RoboDK station: Demo-opstelling - Full - test 2 - for approach point generation - production.rdk

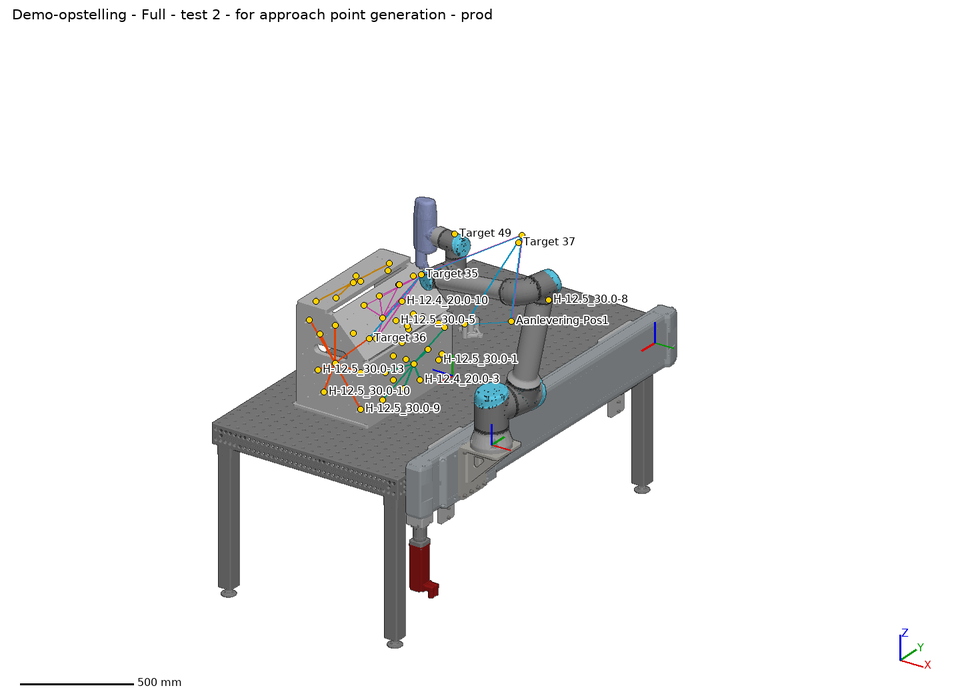
[picture v0: the station drawn from its stored meshes, robots at their saved joint values, targets as dots, program paths as lines]
Station Demo-opstelling - Full - test 2 - Copy (saved by RoboDK 5.9.0). Poses are relative to the parent item; angles as X-Y-Z fixed-axis rotations.
Station parameters (name, value as stored): CollisionFreePlanner, UR10e, CollisionFreePlanner-Rob UR10e, CollisionFreePlanner-Rob My Mechanism, CollisionFreePlanner-Rob Lineaire rail
  - object Lineaire Rail at (0, 0, 0) mm, size 171.1 x 1963 x 635.1 mm
  - object Cobot Carraige at (0, 0, 0) mm, size 240 x 425 x 269.5 mm
  - object Lastafel at (0, 0, 0) mm, size 1021.8 x 2000 x 842 mm
  - frame Lineaire rail  Base at (218.83, 1501.27, 137) mm, rotated rx 0 ry 0 rz -90 deg
    - robot Lineaire rail: 1 axes
        modified DH rows (alpha deg, a mm, theta deg, d mm): 0, 0, 0, 0 linear
        base shift (0, 0, 0) mm, rotated rx 0 ry 90 rz 0 deg
        joint limits [-1248] to [-1248]; home [0]; saved at [-1248]
      - frame UR10e Base at (0, -2, 0.1) mm, rotated rx 0 ry 0 rz 90 deg
        - robot UR10e: 6 axes, payload 10 kg, reach 1300 mm, repeatability 0.05 mm, weight 28.9 kg
            modified DH rows (alpha deg, a mm, theta deg, d mm): 0, 0, 0, 180.7; 90, 0, 180, 0; 0, 612.6, 0, 0; 0, 571.335, 0, 174.15; -90, 0, 0, 119.85; 90, 0, 180, 116.55
            joint limits [100, -200, -360, -480, -360, -360] to [250, 180, 360, 360, 360, 700]; home [30.872, -95.296, 116.362, -22.187, 121.11, 179.827]; saved at [168.209, -76.445, -115.546, 11.991, 92.546, 90.001]
          - tool TCP Schroeftool, TCP at (225, 0, 93) mm, rotated rx 90 ry -90 rz 90 deg, size 86.2 x 125.3 x 346 mm, geometry from Onrobot + custom dop.STEP
          - tool TCP Sensor, TCP at (-192.58, 8.55, 68.16) mm, rotated rx 0 ry -90 rz 0 deg
  - Python program csv_importer_v12 (listed below)
  - program Oppakken (1 instructions, listed below)
  - program indraaien/uitdraaien (1 instructions, listed below)
  - Python program importRobotPoints (listed below)
  - Python program __init__ (listed below)
  - program Prog8 (11 instructions, listed below)
  - frame CSV Frame at (-421.32, 863.78, 53.03) mm, rotated rx 90 ry 0 rz -89.82 deg
    - object Test object at (0, 0, 0) mm, size 650 x 517 x 400 mm, geometry from Test object.STEP
    - target Target 35 (Cartesian target) at (321.7, 636.46, -59.39) mm, rotated rx -90 ry -80.58 rz -180 deg; joints [168.209, -76.49, -91.294, -192.215, -92.546, 270.001] of UR10e
    - target Target 37 (Cartesian target) at (-229.45, 611.91, -197.99) mm, rotated rx 0 ry -0.72 rz 180 deg; joints [123.607, -98.633, -95.414, -165.955, -57.291, 0.002] of UR10e
    - target Target 36 (Cartesian target) at (850.47, 562.22, -149.07) mm, rotated rx 70.72 ry 0 rz -90 deg; joints [244.224, -80.879, -108.983, -80.137, 89.999, 44.77] of UR10e
    - target H-12.5_30.0-0 (Cartesian target) at (10, 165.95, 226.14) mm, rotated rx -90 ry 0 rz -90 deg; joints [161.752, -90.555, -88.742, -182.846, -147.095, -106.726] of UR10e
    - target H-12.5_30.0-1 (Cartesian target) at (10, 61.56, 64.68) mm, rotated rx -90 ry 1.14 rz -90.86 deg; joints [140.207, -149.215, -63.175, -57.939, 88.607, 140.221] of UR10e
    - target H-12.5_30.0-2 (Cartesian target) at (10, 91.63, 261.38) mm, rotated rx -90 ry 0 rz -90 deg; joints [139.629, -149.975, -62.079, -417.947, 89.999, 139.63] of UR10e
    - target H-12.5_30.0-3 (Cartesian target) at (10, 435.06, 200.51) mm, rotated rx -90 ry 0 rz -90 deg; joints [145.332, -190.81, 25.853, -105.043, 89.999, 145.334] of UR10e
    - target H-12.5_30.0-4 (Cartesian target) at (10, 369.06, 279.32) mm, rotated rx -90 ry 0 rz -90 deg; joints [143.714, -169.382, 16.894, 242.486, 89.999, 143.716] of UR10e
    - target H-12.5_30.0-5 (Cartesian target) at (10, 190.3, 292.78) mm, rotated rx -90 ry 0 rz -90 deg; joints [166.618, -153.245, -71.353, -35.667, -87.696, -166.813] of UR10e
    - target H-12.5_30.0-6 (Cartesian target) at (10, 241.56, 64.68) mm, rotated rx -90 ry 0 rz -90 deg; joints [166.782, 132.561, 62.356, 264.825, -87.724, -166.975] of UR10e
    - target H-12.5_30.0-7 (Cartesian target) at (10, 422.89, 336.81) mm, rotated rx -90 ry 0 rz -90 deg; joints [139.629, -141.427, -58.919, -69.655, 89.999, 139.63] of UR10e
    - target H-12.5_30.0-8 (Cartesian target) at (-862.39, -0.19, 81.88) mm, rotated rx 122.16 ry 90 rz -147.65 deg; joints [205.922, -142.466, -64.883, -242.648, -90, -154.261] of UR10e
    - target H-12.5_30.0-9 (Cartesian target) at (610, 61.56, 64.68) mm, rotated rx 90 ry 0 rz -90 deg; joints [202.083, -127.057, -94.792, -48.15, 90, 22.085] of UR10e
    - target H-12.5_30.0-10 (Cartesian target) at (610, 91.63, 261.38) mm, rotated rx 90 ry 0 rz -90 deg; joints [206.662, -125.159, -115.395, -29.445, 89.999, 26.663] of UR10e
    - target H-12.5_30.0-11 (Cartesian target) at (610, 435.06, 200.51) mm, rotated rx 90 ry 0 rz -90 deg; joints [201.283, -134.244, -90.966, -44.789, 90, 21.284] of UR10e
    - target H-12.5_30.0-12 (Cartesian target) at (610, 369.06, 279.32) mm, rotated rx 90 ry 0 rz -90 deg; joints [202.704, -112.114, -87.388, -70.497, 90, 22.705] of UR10e
    - target H-12.5_30.0-13 (Cartesian target) at (610, 190.3, 292.78) mm, rotated rx 90 ry 0 rz -90 deg; joints [200.897, -121.238, -80.649, -68.112, 90, 20.898] of UR10e
    - target H-12.5_30.0-14 (Cartesian target) at (610, 241.56, 64.68) mm, rotated rx 90 ry 0 rz -90 deg; joints [200.617, -130.479, -85.286, -54.234, 90, 20.618] of UR10e
    - target H-12.5_30.0-15 (Cartesian target) at (610, 422.89, 336.81) mm, rotated rx 90 ry 0 rz -90 deg; joints [206.662, -110.651, -112.387, -46.96, 89.999, 26.663] of UR10e
    - target H-12.4_20.0-0 (Cartesian target) at (54.65, 257, 0) mm, rotated rx 0 ry 0 rz -180 deg; joints [173.73, 164.175, 49.241, 18.557, -116.146, -150.598] of UR10e
    - target H-12.4_20.0-1 (Cartesian target) at (530.66, 93.56, 0) mm, rotated rx 0 ry 0 rz -180 deg; joints [158.769, -134.377, -127.415, 81.789, 21.41, -179.996] of UR10e
    - target H-12.4_20.0-2 (Cartesian target) at (510.23, 219.54, 0) mm, rotated rx 0 ry 0 rz -180 deg; joints [221.285, -122.553, -140.995, -96.45, 41.106, 0] of UR10e
    - target H-12.4_20.0-3 (Cartesian target) at (244.64, 75.17, 0) mm, rotated rx 0 ry 0 rz -180 deg; joints [218.989, -104.144, -141.239, -114.615, 38.81, 0] of UR10e
    - target H-12.4_20.0-4 (Cartesian target) at (181.99, 200.48, 0) mm, rotated rx 0 ry 0 rz -180 deg; joints [182.403, -125.392, -139.595, -94.982, 2.224, -0.03] of UR10e
    - target H-12.4_20.0-5 (Cartesian target) at (351.56, 219.54, 0) mm, rotated rx 0 ry 0 rz -180 deg; joints [173.833, -140.994, -133.314, 94.296, 6.346, -179.988] of UR10e
    - target H-12.4_20.0-6 (Cartesian target) at (370.63, 83.35, 0) mm, rotated rx 0 ry 0 rz -180 deg; joints [197.903, -103.418, -142.414, -114.164, 17.724, -0.003] of UR10e
    - target H-12.4_20.0-7 (Cartesian target) at (76.44, 137.14, 0) mm, rotated rx 0 ry 0 rz -180 deg; joints [200.656, -123.841, -142.868, -93.287, 20.477, -0.002] of UR10e
    - target H-12.4_20.0-8 (Cartesian target) at (450.3, 157.57, 0) mm, rotated rx 0 ry 0 rz -180 deg; joints [161.099, -119.903, -130.674, -109.426, -19.079, 360.005] of UR10e
    - target H-12.4_20.0-9 (Cartesian target) at (450.3, 275.38, 0) mm, rotated rx 0 ry 0 rz -180 deg; joints [211.625, -112.452, -143.2, -104.346, 31.446, -0.001] of UR10e
    - target H-12.4_20.0-10 (Cartesian target) at (209.91, 411.7, 119.7) mm, rotated rx 18.88 ry -41.64 rz 62.76 deg; joints [149.478, -123.359, -101.972, -255.509, 129.295, 117.809] of UR10e
    - target H-12.4_20.0-11 (Cartesian target) at (425.79, 464.67, 172.67) mm, rotated rx 32.73 ry -32.8 rz 40.12 deg; joints [165.417, -91.386, -120.357, -91.866, 220.573, -73.917] of UR10e
    - target H-12.4_20.0-12 (Cartesian target) at (489.8, 356.81, 64.81) mm, rotated rx 0.56 ry -45 rz 89.21 deg; joints [187.536, -115.219, -134.443, -245.153, 85.362, -275.211] of UR10e
    - target H-12.4_20.0-13 (Cartesian target) at (309.34, 464.67, 172.67) mm, rotated rx 26.57 ry -37.76 rz 50.77 deg; joints [157.394, -95.698, -117.978, -87.531, 225.724, -67.512] of UR10e
    - target H-12.4_20.0-14 (Cartesian target) at (163.61, 461.3, 169.3) mm, rotated rx 18.88 ry -41.64 rz 62.76 deg; joints [148.298, -102.262, -112.081, -85.655, 230.107, -60.871] of UR10e
    - target H-12.4_20.0-15 (Cartesian target) at (159.52, 338.03, 46.03) mm, rotated rx 45 ry 0 rz 0 deg; joints [148.298, -102.262, -112.081, -85.655, 230.107, -60.871] of UR10e
    - target H-12.4_20.0-16 (Cartesian target) at (275.97, 338.03, 46.03) mm, rotated rx 45 ry 0 rz 0 deg; joints [140.381, -117.925, -81.399, -160.677, 140.203, -135] of UR10e
    - target H-12.4_20.0-17 (Cartesian target) at (589.22, 408.81, 116.81) mm, rotated rx 40.89 ry -20.7 rz 22.21 deg; joints [147.265, -110.05, -92.953, -156.998, 147.087, -135] of UR10e
    - target H-12.4_20.0-18 (Cartesian target) at (72.35, 497, 283.1) mm, rotated rx 90 ry -80 rz 0 deg; joints [176.842, -85.894, -126.259, -98.403, 207.733, -84.925] of UR10e
    - target H-12.4_20.0-19 (Cartesian target) at (261.67, 497, 331.45) mm, rotated rx 90 ry -50 rz 0 deg; joints [152.167, -171.826, 50.873, 120.952, 231.99, -89.999] of UR10e
    - target H-12.4_20.0-20 (Cartesian target) at (487.76, 497, 279.01) mm, rotated rx 90 ry -76.62 rz 0 deg; joints [180.252, -108.499, -96.736, 25.234, 103.309, -269.999] of UR10e
    - target H-12.4_20.0-21 (Cartesian target) at (567.43, 497, 331.45) mm, rotated rx 90 ry -75.8 rz 0 deg; joints [186.047, -111.869, -91.994, 23.863, 98.334, -269.999] of UR10e
    - target H-12.4_20.0-22 (Cartesian target) at (292.31, 497, 283.1) mm, rotated rx 90 ry -50 rz 0 deg; joints [176.725, -122.81, -75.29, 18.1, 153.453, -269.999] of UR10e
    - target Target 49 (Cartesian target) at (377.54, 920.16, -278.05) mm, rotated rx -90 ry -64.33 rz -180 deg; joints [191.308, -67.601, -62.99, -229.408, -53.196, 270.001] of UR10e
    - target Face_Target_1_0_0 (Cartesian target) at (10, 248.31, 200.75) mm, rotated rx -90 ry 0 rz -90 deg; joints [211.342, -122.635, -119.421, -27.943, 89.999, 31.169] of UR10e
    - target Face_Target_-1_0_0 (Cartesian target) at (610, 248.31, 200.75) mm, rotated rx 90 ry 0 rz -90 deg; joints [211.342, -122.635, -119.421, -27.943, 89.999, 31.169] of UR10e
    - target Face_Target_0_0_1 (Cartesian target) at (292.65, 175.28, 0) mm, rotated rx 0 ry 0 rz -180 deg; joints [211.342, -122.635, -119.421, -27.943, 89.999, 31.169] of UR10e
    - target Face_Target_0_-1_1 (Cartesian target) at (374.37, 401.35, 109.35) mm, rotated rx 18.88 ry -41.64 rz 62.76 deg; joints [164.138, -116.912, -117.695, 105.295, 120.817, 103.152] of UR10e
    - target Face_Target_0_-1_0 (Cartesian target) at (319.89, 497, 305.23) mm, rotated rx 90 ry -80 rz 0 deg; joints [211.342, -122.635, -119.421, -27.943, 89.999, 31.169] of UR10e
    - target Target 49 (Cartesian target) at (292.65, 175.28, 0) mm, rotated rx 0 ry 0 rz -180 deg; joints [189.308, -110.392, -141.765, -107.836, 9.129, -0.006] of UR10e
    - target Target 50 (Cartesian target) at (610, 248.31, 200.75) mm, rotated rx 90.01 ry 0 rz -90 deg; joints [206.665, -136.526, -67.038, -246.438, -89.999, 206.493] of UR10e
    - target Target 37 new (Cartesian target) at (-205.62, 667.37, -232.74) mm, rotated rx -1.98 ry 0.78 rz -89.43 deg; joints [114.4, -103.093, -74.88, -92.872, 89.521, 202.246] of UR10e
    - object Assem- houder (1) at (-379.38, 0, -15.78) mm, rotated rx 0 ry 0 rz 90 deg, geometry from Assem- houder (1).STEP
      - item type 7 Assem- houder (1)-0
        - item type 7 Assem- houder (1)-0-0
        - item type 7 Assem- houder (1)-0-1
        - item type 7 Assem- houder (1)-0-2
        - item type 7 Assem- houder (1)-0-3
        - item type 7 Assem- houder (1)-0-4
        - item type 7 Assem- houder (1)-0-5
        - item type 7 Assem- houder (1)-0-6
        - item type 7 Assem- houder (1)-0-7
        - item type 7 Assem- houder (1)-0-8
        - item type 7 Assem- houder (1)-0-9
        - item type 7 Assem- houder (1)-0-10
        - item type 7 Assem- houder (1)-0-11
        - item type 7 Assem- houder (1)-0-12
        - item type 7 Assem- houder (1)-0-13
        - item type 7 Assem- houder (1)-0-14
        - item type 7 Assem- houder (1)-0-15
        - item type 7 Assem- houder (1)-0-16
        - item type 7 Assem- houder (1)-0-17
        - item type 7 Assem- houder (1)-0-18
        - item type 7 Assem- houder (1)-0-19
        - item type 7 Assem- houder (1)-0-20
        - item type 7 Assem- houder (1)-0-21
        - item type 7 Assem- houder (1)-0-22
      - item type 7 Assem- houder (1)-1
    - object Toolswitch M5 M8 M12 at (-389.95, 0, 108.57) mm, size 112.6 x 60.1 x 126.6 mm, geometry from Toolswitch M5 M8 M12.STEP
    - target Aanlevering-Pos1 (Cartesian target) at (-389.05, 120.04, -45.2) mm, rotated rx -175.62 ry -49.73 rz -92.03 deg; joints [128.562, 159.009, 53.75, -85.478, 125.727, 54.228] of UR10e
    - target Toolswitch-m8 (Cartesian target) at (-344.01, 65.34, 170.68) mm, rotated rx -90 ry -60.73 rz 180 deg; joints [135.813, -158.432, -55.566, 33.999, -254.903, 450.001] of UR10e
  - program Prog9 (12 instructions, listed below)
  - Python program ProgramGenerator (listed below)
    - Python program ProgramGenerator (listed below)
  - Python program csv_importer (listed below)
  - Python program csv_importernewest (listed below)
  - Python program Make_approaches_paths (listed below)
  - Python program TargetFixer (listed below)
  - Python program generatefaceapproaches (listed below)
  - Python program csvimporterLauranewest (listed below)
  - Python program Addmoveshanktoprog (listed below)
  - program Prog20 (14 instructions, listed below)
  - program Program_Face_-1_0_0 (19 instructions, listed below)
  - program Program_Face_0_0_1 (17 instructions, listed below)
  - program Program_Face_0_-1_1 (54 instructions, listed below)
  - program Program_Face_0_-1_0 (13 instructions, listed below)
  - program Prog22 (12 instructions, listed below)
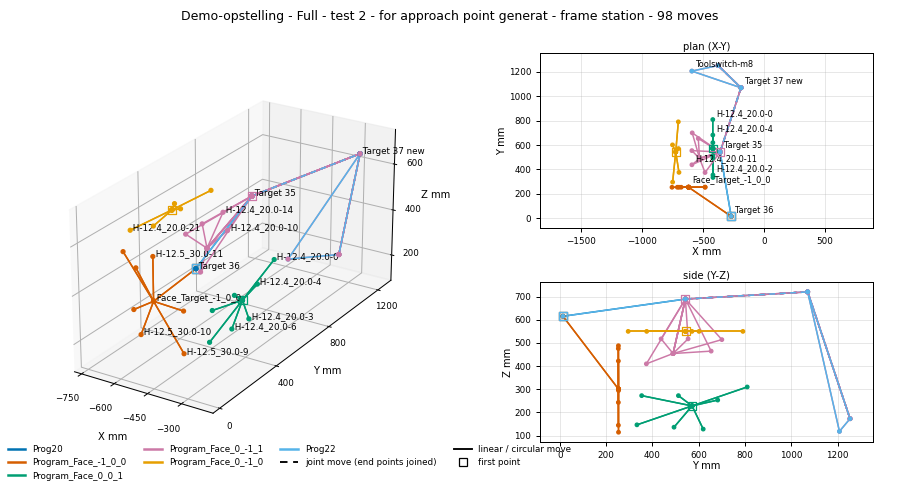
[picture p0: tool path of Demo-opstelling - Full - test 2 - for approach point generation - production.rdk in frame station, 98 of 117 moves have a stored position in this frame; points joined in program order, loops and branches not executed]

--- Python program csv_importer_v12 ---
# This macro can load CSV files from Denso programs in RoboDK.
# Supported types of files are:
#  1-Tool data : Tool.csv
#  2-Work object data: Work.csv
#  3-Target data: P_Var.csv
# This macro can also filter a given targets file

# Type help("robodk.robolink") or help("robodk.robomath") for more information
# Press F5 to run the script
# Visit: http://www.robodk.com/doc/PythonAPI/
# For RoboDK API documentation

import os
import datetime

import tkinter as tk
from tkinter import messagebox

from robodk.robolink import *  # API to communicate with RoboDK
from robodk.robomath import *  # Robot toolbox
from robodk.robodialogs import *
from robodk.robofileio import *
import robodk.robolinkutils as RDKutils

DEBUG = False

debuglist = []

# Start communication with RoboDK
RDK = Robolink()

# Ask the user to select the robot
ROBOT = RDK.ItemUserPick('Select a robot', ITEM_TYPE_ROBOT)

# Check if the user selected a robot
if not ROBOT.Valid():
    quit()


# Ask the user to select a reference frame and get the active tool
BASE = ROBOT.Parent()
#BASE = RDK.Item('UR10e Base', ITEM_TYPE_FRAME)
#BASE = RDK.ItemUserPick('Select robot base frame', ITEM_TYPE_FRAME)
FRAME = RDK.ItemUserPick('Reference Frame', ITEM_TYPE_FRAME)
FRAMEPOSE = RDKutils.getPoseWrt(FRAME, BASE) #frame pose wrt robot base
TOOL = ROBOT.getLink(ITEM_TYPE_TOOL)
TOOLPOSE = RDKutils.getPoseWrt(TOOL, TOOL.Parent()) #tool pose wrt robot flange

if not FRAME.Valid() or not TOOL.Valid():
    raise Exception("Select appropriate FRAME and TOOL references")


# Function to convert XYZWPR to a pose
# Important! Specify the order of rotation
def xyzwpr_to_pose(xyzwpr):
    x, y, z, rx, ry, rz = xyzwpr
    return point_Zaxis_2_pose([x, y, z], [-rx, -ry, -rz])
    #return transl(x, y, z) * rotz(rz * pi / 180) * roty(ry * pi / 180) * rotx(rx * pi / 180)
    #return transl(x,y,z)*rotx(rx*pi/180)*roty(ry*pi/180)*rotz(rz*pi/180)
    #return KUKA_2_Pose(xyzwpr)


# csv_file = 'C:/Users/Albert/Desktop/Var_P.csv'
csv_file = getOpenFileName(RDK.getParam('PATH_OPENSTATION'))

# Specify file codec
codec = 'utf-8'  #'ISO-8859-1'


# Load P_Var.CSV data as a list of poses, including links to reference and tool frames
def load_targets(strfile):
    csvdata = LoadList(strfile, ',', codec)
    poses = []
    idxs = []
    for i in range(0, len(csvdata)):
        x, y, z, rx, ry, rz = csvdata[i][0:6]
        poses.append(xyzwpr_to_pose([x, y, z, rx, ry, rz]))
        #idxs.append(csvdata[i][6])
        idxs.append(i)

    return poses, idxs


# Load and display Targets from P_Var.CSV in RoboDK
def make_targets(strfile):
    poses, idxs = load_targets(strfile)
    program_name = getFileName(strfile)
    program_name = program_name.replace('-', '_').replace(' ', '_')

    for pose, idx in zip(poses, idxs):
        name = 'H-%s-%i' % (program_name, idx)
        target = RDK.Item(name, ITEM_TYPE_TARGET)
        if target.Valid():
            target.Delete()
        target = RDK.AddTarget(name, FRAME, ROBOT)
        target.setPose(pose)
        collision_free(target, idx)

def test_all_configurations(configurations):
    for joints in configurations:

        # turn collision checking off
        RDK.setCollisionActive(COLLISION_OFF)
        if DEBUG:
            is_active = RDK.Command("CollisionActive")
            print(f"collsion active? should be off (0) {is_active}")
            debuglist.append(f"collsion active? should be off (0) {is_active}")

        # move to target
        try:
            ROBOT.MoveJ(joints)
        except TargetReachError:
            continue

        # turn collision checking on, test for collisions
        RDK.setCollisionActive(COLLISION_ON)
        if DEBUG:
            is_active = RDK.Command("CollisionActive")
            print(f"collsion active? should be on (1) {is_active}")
            debuglist.append(f"collsion active? should be on (1) {is_active}")

        collision = RDK.Collisions()
        if DEBUG:
            print(f"collision: {collision}")
            debuglist.append(f"collision: {collision}")

        collision_items = RDK.CollisionItems()
        if TOOL in collision_items or collision == 0:
            break

    try:
        collision
    except NameError:
        collision = -2
        if DEBUG:
            print("Target cannot be reached or is to close to a singularity")
            debuglist.append("Target cannot be reached or is to close to a singularity")

    return collision


def test_collision_target(target, rz):
    if DEBUG:
        print("testing at target")
        debuglist.append("testing at target")

    possible_robot_configurations = ROBOT.SolveIK_All(target.Pose(), tool=TOOLPOSE, reference=FRAMEPOSE)
    issues_value = test_all_configurations(possible_robot_configurations) # returns 0 if at least one configuration is without issues

    return issues_value

def test_issues_point(target, rz):
    if DEBUG:
        print("testing point")
        debuglist.append("testing point")

    # define the rotated position to test for collisions
    target_new_pose = RelTool(target.Pose(), 0,0,0, 0,0,rz)
    possible_robot_configurations = ROBOT.SolveIK_All(target_new_pose, tool=TOOLPOSE, reference=FRAMEPOSE)
    issues_value = test_all_configurations(possible_robot_configurations) # returns 0 if at least one configuration is without issues

    return issues_value, target_new_pose

rotation_direction = "pos"
direction_changes = 0
holes_no_solution = []

def collision_free(target, idx):
    rotation_step = 10
    repmax = 360/rotation_step
    global rotation_direction
    global direction_changes
    s = 0
    rep = 0
    if DEBUG:
        print(f"\nHole {idx}")
        debuglist.append(f"\nHole {idx}")

    issues_value, target_new_pose = test_issues_point(target, 0)
    if DEBUG:
        print(f"issues value: {issues_value}")
        debuglist.append(f"issues value: {issues_value}")

    while issues_value != 0 and s < 100: # s for safety, so it can't go on forever
        if DEBUG:
            print(f"s before: {s}")
            debuglist.append(f"s before: {s}")
            print(f"rep: {rep}")
            debuglist.append(f"rep: {rep}")
            print(f"rotation direction: {rotation_direction}")
            debuglist.append(f"rotation direction: {rotation_direction}")
            print(f"direction changes: {direction_changes}")
            debuglist.append(f"direction changes: {direction_changes}")

        s += 1

        if issues_value == -2 and direction_changes < 2:
			#target unreachable
            if rotation_direction == "pos":
                rotation_direction = "neg"
                direction_changes += 1
                r = -1 #rotation factor to make the rotation negative
            else:
                rotation_direction = "pos"
                direction_changes += 1
                r = 1 #rotation factor to make the rotation positive
            issues_value, target_new_pose = test_issues_point(target, r*rotation_step)
            target.setPose(target_new_pose)

        elif issues_value > 0 and rep < repmax:
			#collision
            RDK.setCollisionActive(COLLISION_OFF)
            if DEBUG:
                is_active = RDK.Command("CollisionActive")
                print(f"collsion active? should be off (0) {is_active}")
                debuglist.append(f"collsion active? should be off (0) {is_active}")

            ROBOT.MoveJ(target.Pose())
            if rotation_direction == "neg":
                r = -1
            elif rotation_direction == "pos":
                r = 1
            issues_value, target_new_pose = test_issues_point(target, r*rotation_step)
            target.setPose(target_new_pose)
            rep += 1

        elif direction_changes >= 2 or rep >= repmax:
            break

        else:
            RDK.ShowMessage(f"Unknown error occured at Hole {idx} while looking for collision free position")
            if DEBUG:
                print(f"Unknown error occured at Hole {idx} while looking for collision free position")
                debuglist.append(f"Unknown error occured at Hole {idx} while looking for collision free position")

    direction_changes = 0
    if issues_value == 0:
        print(f"No issues at Hole {idx}")
        debuglist.append(f"No issues at Hole {idx}")
    elif direction_changes >= 2 or rep >= repmax or s >= 100:
        RDK.ShowMessage(f"No solution found for Hole {idx}", False)
        holes_no_solution.append(idx)
        if DEBUG:
            print(f"No solution found for Hole {idx}")
            debuglist.append(f"No solution found for Hole {idx}")
    else:
        RDK.ShowMessage(f"Unknown error occured at Hole {idx} while looking for collision free position")
        if DEBUG:
            print(f"Unknown error occured at Hole {idx} while looking for collision free position")
            debuglist.append(f"Unknown error occured at Hole {idx} while looking for collision free position")


MAKE_GUI_PROGRAM = True

ROBOT.setFrame(FRAME)
ROBOT.setTool(TOOL)

if RDK.RunMode() == RUNMODE_SIMULATE:
    MAKE_GUI_PROGRAM = True
    # MAKE_GUI_PROGRAM = mbox('Do you want to create a new program? If not, the robot will just move along the targets', 'Yes', 'No')
else:
    # if we run in program generation mode just move the robot
    MAKE_GUI_PROGRAM = False

if MAKE_GUI_PROGRAM:
    RDK.Render(False)  # Faster if we turn render off
    make_targets(csv_file)
else:
    l

RDK.ShowMessage(f"Holes without solution: {holes_no_solution}")

if DEBUG:
    print(f"Holes without solution: {holes_no_solution}")
    debuglist.append(f"Holes without solution: {holes_no_solution}")

    current_time = datetime.datetime.now()
    filename = os.path.splitext(os.path.basename(__file__))
    with open("C:/Users/Laura/Documents/1.Windesheim/Stage/2024/Lectoraat/Deelvragen/2.Targets maken/debugfile.txt", "a") as file:
        file.write("\n\n-----------------------------------------------\n")
        file.write(current_time.strftime("%c"))
        file.write("\n-----------------------------------------------\n")
        for prints in debuglist:
            file.write(prints)
            file.write("\n")
        file.write(holes_no_solution)
        file.write(filename[0])

--- program Oppakken (robot UR10e) ---
  sd_move(23,0)
      se...: sd_move(23,0)
      set_digital_out(1, True)
      sleep(0.025)
      force_mode(tool_pose(), [0, 0, 1, 0, 0, 0], [0.0, 0.0, -2.0, 0.0, 0.0, 0.0], 2, [0.1, 0.1, 0.15, 0.17, 0.17, 0.17])
      sd_tighten(0, 20, 1, 0)
      sleep(3)
      end_force_mode()
      sd_stop(0)
      set_digital_out(1, False)
      sleep(0.5)
      sd_move(0,0 )

--- program indraaien/uitdraaien (robot UR10e) ---
  sd_move(23,0)
      sleep(0.025)
      force_mode(tool_pose(), [0, 0, 1, 0, 0, 0], [0.0, 0.0, -10.0, 0.0, 0.0, 0.0], 2, [0.1, 0.1, 0.15, 0.17, 0.17, 0.17])
      sd_tighten(0, 30, 1, 0)
      sleep(1)
      end_force_mode()
      
      sleep(0.025)
      freedrive_mode([1, 1, 1, 0, 0, 0], tool_pose())
      sd_move(55,0)
      sd_loosen(-2, 50, 0)
      sleep(5)
      sd_move(0, 0)
      end_freedrive_mode()
      sd_stop(0)

--- Python program importRobotPoints ---
#-----
#Import Robot Points
#
#Import data in csv as motion statements into robot program.
#-----
#Version 1.0
#-----
#CSV file can have the following fields (in any order dictated by the first line) where only X,Y,Z are mandatory:
#
#Name,X,Y,Z,RX,RY,RZ,Base,Tool,Motion,MaxSpeed,JointSpeed,AccuracyValue,E1,E2,E3,E4,E5,E6
#P1,100.0,200.0,300.0,0,90,0,Base1,Gripper,LIN,1000.0,100.0,5.0,111.1,222.2,0,0,0,0
#-----

from vcCommand import *
import vcMatrix, vcVector

app = getApplication()
cmd = getCommand()
#-----
def OnStart():
  rou = app.TeachContext.ActiveRoutine
  if not rou:
    print 'No robot selected.'
    return

  open_dialog = app.findCommand('dialogOpen')
  open_dialog.OnPostExecute = readCSV
  open_dialog.Param_3 = 'CSV Files (*.csv)|*.csv'
  open_dialog.execute()
#-----
def readCSV(open_dialog):
  open_dialog.OnPostExecute = None
  uri = open_dialog.Param_1[8:]

  rou = app.TeachContext.ActiveRoutine
  exe = rou.Program.Executor
  ctr = exe.Controller
  mt_init = ctr.createTarget()
  separator = ','

  with open(uri, 'r') as csv_file:

    #Try to find separator character from first line
    line = csv_file.readline()
    line = line.rstrip('\n')
    line = line.lower()
    count = 0
    trythese = ',;:'
    for c in trythese:
      if line.count(c) > count:
        count = line.count(c)
        separator = c
      #endif
    #endfor

    #Find out data headers on the first line
    fields = line.split(separator)
    if not 'x' in fields or not 'y' in fields or not 'z' in fields:
      #No coordinate data (only necessary fields)
      print 'No XYZ data found in the header. Aborting.'
      return

    #Iterate data lines
    index = 0
    for line in csv_file:
      index +=1

      line = line.rstrip('\n')
      data = line.split(separator)

      name = 'P' + str(index)
      x = 0
      y = 0
      z = 0
      w = 0
      p = 0
      r = 0
      base = getBase(ctr,mt_init.BaseName)
      tool = getTool(ctr,mt_init.ToolName)
      motion = VC_STATEMENT_LINMOTION
      max_speed = 1000.0
      joint_speed = 1.0
      accuracy = 0.0
      ex_joints = []

      try:
        x = float(data[fields.index('x')])
        y = float(data[fields.index('y')])
        z = float(data[fields.index('z')])

        if 'name' in fields:
          name = data[fields.index('name')]

        if 'rx' in fields and 'ry' in fields and 'rz' in fields:
          w = float(data[fields.index('rx')])
          p = float(data[fields.index('ry')])
          r = float(data[fields.index('rz')])
        elif 'w' in fields and 'p' in fields and 'r' in fields:
          w = float(data[fields.index('w')])
          p = float(data[fields.index('p')])
          r = float(data[fields.index('r')])
        elif 'a' in fields and 'b' in fields and 'c' in fields:
          #A=RZ, B=RY, C=RX
          w = float(data[fields.index('c')])
          p = float(data[fields.index('b')])
          r = float(data[fields.index('a')])

        if 'base' in fields:
          base = getBase(ctr,data[fields.index('base')])
        if 'tool' in fields:
          tool = getTool(ctr,data[fields.index('tool')])

        if 'motion' in fields:
          if data[fields.index('motion')].lower() == 'ptp':
            motion = VC_STATEMENT_PTPMOTION

        if 'maxspeed' in fields:
          max_speed = float(data[fields.index('maxspeed')])

        if 'jointspeed' in fields:
          joint_speed = float(data[fields.index('jointspeed')]) / 100.0

        if 'accuracyvalue' in fields:
          accuracy = float(data[fields.index('accuracyvalue')])

        for i in range(6):
          e_name = 'e' + str(i+1)
          if e_name in fields:
            ex_joints.append(float(data[fields.index(e_name)]))

      except:
        print 'Invalid data line, skipping.'
        continue

      m = vcMatrix.new()
      m.translateAbs(x,y,z)
      m.setWPR(w,p,r)

      stat = rou.addStatement(motion)
      stat.readIn()
      stat.Positions[0].Name = name
      stat.Positions[0].PositionInReference = m
      stat.Base = base
      stat.Tool = tool
      stat.AccuracyMethod = VC_MOTIONTARGET_AM_DISTANCE
      stat.AccuracyValue = accuracy

      if motion == VC_STATEMENT_LINMOTION:
        stat.MaxSpeed = max_speed
      else:
        stat.JointSpeed = joint_speed



      for i in range(len(ex_joints)):
        e_name = 'E' + str(i+1)
        prop = stat.Positions[0].getProperty(e_name)
        if prop:
          prop.Value = ex_joints[i]
    #endfor line in csv_file:
  #endwith open(uri, 'r') as csv_file:

  app.render()
  print 'Done.'
#-----
def getBase(ctr, base_name):
  for base in ctr.Bases:
    if base.Name == base_name:
      return base
  return None
#-----
def getTool(ctr, tool_name):
  for tool in ctr.Tools:
    if tool.Name == tool_name:
      return tool
  return None
#-----

--- Python program __init__ ---
#-----
#Import Robot Points init
#
#Import data in csv as motion statements into robot program.
#-----
#Version 1.0
#-----
from vcApplication import *

def OnStart():
  cmduri = getApplicationPath() + 'importRobotPoints.py'
  cmd = loadCommand('ImportRobotPoints',cmduri)
  addMenuItem('VcTabTeach/Import', "Import CSV", -1, "ImportRobotPoints")

--- program Prog8 (robot UR10e) ---
  Set Ref.: CSV Frame
  Set Tool: TCP Schroeftool
  MoveJ (H-10.2_30.0-1) [its target is no longer in the station]
  MoveJ (H-10.2_30.0-2) [its target is no longer in the station]
  MoveJ (H-10.2_30.0-3) [its target is no longer in the station]
  MoveJ (H-10.2_30.0-4) [its target is no longer in the station]
  MoveJ (H-10.2_30.0-5) [its target is no longer in the station]
  MoveJ (H-10.2_30.0-6) [its target is no longer in the station]
  MoveJ (H-10.2_30.0-7) [its target is no longer in the station]
  MoveJ (H-10.2_30.0-8) [its target is no longer in the station]
  MoveJ (H-10.2_30.0-9) [its target is no longer in the station]

--- program Prog9 (robot UR10e) ---
  Set Ref.: CSV Frame
  Set Tool: TCP Schroeftool
  MoveJ (H-10.2_30.0.csv-0) [its target is no longer in the station]
  MoveJ (H-10.2_30.0.csv-1) [its target is no longer in the station]
  MoveJ (H-10.2_30.0.csv-2) [its target is no longer in the station]
  MoveJ (H-10.2_30.0.csv-3) [its target is no longer in the station]
  MoveJ (H-10.2_30.0.csv-4) [its target is no longer in the station]
  MoveJ (H-10.2_30.0.csv-5) [its target is no longer in the station]
  MoveJ (H-10.2_30.0.csv-6) [its target is no longer in the station]
  MoveJ (H-10.2_30.0.csv-7) [its target is no longer in the station]
  MoveJ (H-10.2_30.0.csv-8) [its target is no longer in the station]
  MoveJ (H-10.2_30.0.csv-9) [its target is no longer in the station]

--- Python program ProgramGenerator ---
from robodk import robolink

# Connect to RoboDK
RDK = robolink.Robolink()

# Get the robot, reference frame, and base point
robot = RDK.Item('UR10e')  # Replace 'Robot' with your robot's name
reference_frame = RDK.Item('CSV Frame')  # Replace 'Reference Frame' with your frame's name
base_point = RDK.Item('Target 33')  # Replace 'Point 1' with your base point's name

# Create a new program
program = RDK.AddProgram('AutoProgram')

# Get all targets under the reference frame
targets = reference_frame.Childs()
target_list = [target for target in targets if target.Type() == robolink.ITEM_TYPE_TARGET]

# Add movements and screwdriver actions to the program
for i, target in enumerate(target_list):
    # Move to the base point first (except for the first target)
    if i > 0:
        program.MoveL(base_point)

    # Move to the target point
    program.MoveL(target)

    # Execute screwdriver actions
    program.RunInstruction('move_shank(20)', robolink.INSTRUCTION_CALL_PROGRAM)  # Tighten screw
    program.RunInstruction('move_shank(0)', robolink.INSTRUCTION_CALL_PROGRAM)  # Release screwdriver

# Save the program
#program.ShowTargets(False)  # Hide targets for clarity
program.Update()
print("Program generated successfully!")

--- Python program ProgramGenerator ---
from robodk import robolink

# Connect to RoboDK
RDK = robolink.Robolink()

# Get the robot, reference frame, and base point
robot = RDK.Item('UR10e')  # Replace 'Robot' with your robot's name
reference_frame = RDK.Item('CSV Frame')  # Replace 'Reference Frame' with your frame's name
base_point = RDK.Item('Target 33')  # Replace 'Point 1' with your base point's name

# Create a new program
program = RDK.AddProgram('AutoProgram')

# Get all targets under the reference frame
targets = reference_frame.Childs()
target_list = [target for target in targets if target.Type() == robolink.ITEM_TYPE_TARGET]

# Add movements and screwdriver actions to the program
for i, target in enumerate(target_list):
    # Move to the base point first (except for the first target)
    if i > 0:
        program.MoveL(base_point)

    # Move to the target point
    program.MoveL(target)

    # Execute screwdriver actions
    program.RunInstruction('move_shank(20)', robolink.INSTRUCTION_CALL_PROGRAM)  # Tighten screw
    program.RunInstruction('move_shank(0)', robolink.INSTRUCTION_CALL_PROGRAM)  # Release screwdriver

# Save the program
#program.ShowTargets(False)  # Hide targets for clarity
program.Update()
print("Program generated successfully!")

--- Python program csv_importer ---
# This macro can load CSV files from Denso programs in RoboDK.
# Supported types of files are:
#  1-Tool data : Tool.csv
#  2-Work object data: Work.csv
#  3-Target data: P_Var.csv
# This macro can also filter a given targets file

# Type help("robodk.robolink") or help("robodk.robomath") for more information
# Press F5 to run the script
# Visit: http://www.robodk.com/doc/PythonAPI/
# For RoboDK API documentation

import os
import datetime

import tkinter as tk
from tkinter import messagebox

from robodk.robolink import *  # API to communicate with RoboDK
from robodk.robomath import *  # Robot toolbox
from robodk.robodialogs import *
from robodk.robofileio import *
import robodk.robolinkutils as RDKutils

DEBUG = False

debuglist = []

# Start communication with RoboDK
RDK = Robolink()

# Ask the user to select the robot
ROBOT = RDK.ItemUserPick('Select a robot', ITEM_TYPE_ROBOT)

# Check if the user selected a robot
if not ROBOT.Valid():
    quit()


# Ask the user to select a reference frame and get the active tool
BASE = ROBOT.Parent()
#BASE = RDK.Item('UR10e Base', ITEM_TYPE_FRAME)
#BASE = RDK.ItemUserPick('Select robot base frame', ITEM_TYPE_FRAME)
FRAME = RDK.ItemUserPick('Reference Frame', ITEM_TYPE_FRAME)
FRAMEPOSE = RDKutils.getPoseWrt(FRAME, BASE) #frame pose wrt robot base
TOOL = ROBOT.getLink(ITEM_TYPE_TOOL)
TOOLPOSE = RDKutils.getPoseWrt(TOOL, TOOL.Parent()) #tool pose wrt robot flange

if not FRAME.Valid() or not TOOL.Valid():
    raise Exception("Select appropriate FRAME and TOOL references")


# Function to convert XYZWPR to a pose
# Important! Specify the order of rotation
def xyzwpr_to_pose(xyzwpr):
    x, y, z, rx, ry, rz = xyzwpr
    return point_Zaxis_2_pose([x, y, z], [-rx, -ry, -rz])



# csv_file = 'C:/Users/Albert/Desktop/Var_P.csv'
csv_file = getOpenFileName(RDK.getParam('PATH_OPENSTATION'))

# Specify file codec
codec = 'utf-8'  #'ISO-8859-1'

def mirror_target(xyzwpr):
    """
    Mirrors the target position and adjusts the rotation.
    Assumes the wall is aligned with the YZ plane (mirroring the X coordinate).
    """
    x, y, z, rx, ry, rz = xyzwpr

    # Mirror the position (reflect across the YZ plane)
    x_mirrored = x  # Negate the X coordinate
    y_mirrored = y   # Keep Y and Z the same
    z_mirrored = z

    # Adjust the rotation (flip RX and RZ)
    rx_mirrored = rx  # Negate RX
    ry_mirrored = ry   # Keep RY the same
    rz_mirrored = -rz  # Negate RZ

    return [x_mirrored, y_mirrored, z_mirrored, rx_mirrored, ry_mirrored, rz_mirrored]

def load_targets(strfile):
    csvdata = LoadList(strfile, ',', codec)
    poses = []
    idxs = []
    for i in range(0, len(csvdata)):
        x, y, z, rx, ry, rz = csvdata[i][0:6]

        # Mirror the target
        x_mirrored, y_mirrored, z_mirrored, rx_mirrored, ry_mirrored, rz_mirrored = mirror_target([x, y, z, rx, ry, rz])

        # Convert the mirrored target to a pose
        poses.append(xyzwpr_to_pose([x_mirrored, y_mirrored, z_mirrored, rx_mirrored, ry_mirrored, rz_mirrored]))
        idxs.append(i)
    return poses, idxs


# Load and display Targets from P_Var.CSV in RoboDK
def make_targets(strfile):
    """Load and display Targets from P_Var.CSV in RoboDK with robust error handling."""
    # Initialize empty lists to collect results
    poses, idxs = load_targets(strfile)
    program_name = getFileName(strfile)
    program_name = program_name.replace('-', '_').replace(' ', '_')

    holes_no_solution = []
    total_targets = len(poses)
    processed_targets = 0

    # Show progress message
    RDK.ShowMessage(f"Processing {total_targets} targets...", False)

    # Process each target
    for pose, idx in zip(poses, idxs):
        try:
            processed_targets += 1
            if processed_targets % 5 == 0:  # Update progress every 5 targets
                RDK.ShowMessage(f"Processing target {processed_targets} of {total_targets}...", False)

            name = 'H-%s-%i' % (program_name, idx)

            # Check if target already exists and delete it
            target = RDK.Item(name, ITEM_TYPE_TARGET)
            if target.Valid():
                target.Delete()

            # Create new target and set pose
            target = RDK.AddTarget(name, FRAME, ROBOT)
            target.setPose(pose)

            # Try to find a collision-free configuration
            if not find_collision_free_configuration(target, idx):
                holes_no_solution.append(idx)
                if DEBUG:
                    print(f"No solution for Hole {idx}")
                    debuglist.append(f"No solution for Hole {idx}")

        except Exception as e:
            # Log error but continue with next target
            holes_no_solution.append(idx)
            if DEBUG:
                print(f"Error processing Hole {idx}: {e}")
                debuglist.append(f"Error processing Hole {idx}: {e}")

    # Show completion message
    if holes_no_solution:
        RDK.ShowMessage(f"Completed with {len(holes_no_solution)} targets without solution: {holes_no_solution}", False)
    else:
        RDK.ShowMessage("All targets processed successfully!", False)

    return holes_no_solution

def test_collision_safe(pose, test_move=False):
    """
    Test a pose for collisions without triggering script interruption.

    Args:
        pose: The pose to test
        test_move: Whether to actually move the robot (False = calculate only)

    Returns:
        0: No collision detected
        1: Collision detected
        -2: Pose unreachable
    """
    # Turn off collision detection while we test
    RDK.setCollisionActive(COLLISION_OFF)

    try:
        # Check if the pose is reachable without moving
        joints = ROBOT.SolveIK(pose, TOOLPOSE, FRAMEPOSE)

        if joints is None or len(joints) == 0:
            return -2  # Unreachable

        if test_move:
            # Try moving to the position with collisions off
            try:
                ROBOT.MoveJ(joints)
            except:
                return -2  # Problem moving, treat as unreachable

        # Check collision after positioning but without movement
        # This allows us to check without triggering interruption
        RDK.setCollisionActive(COLLISION_ON)
        collision = RDK.Collisions()

        if collision > 0:
            return 1  # Collision detected
        else:
            return 0  # No collision

    except Exception as e:
        if DEBUG:
            print(f"Error in collision testing: {e}")
            debuglist.append(f"Error in collision testing: {e}")
        return -2  # Any error, treat as unreachable

    finally:
        # Always make sure we turn collision checking back off
        RDK.setCollisionActive(COLLISION_OFF)


def test_all_configurations(configurations):
    """Test all robot configurations and find one without collisions.
    Returns:
        0: If a collision-free configuration is found
        1: If all configurations have collisions
        -2: If no configurations are reachable
    """
    if not configurations:
        return -2  # No configurations available

    for joints in configurations:
        # Turn collision checking off for movement
        RDK.setCollisionActive(COLLISION_OFF)

        # Try to move to target configuration with error handling
        try:
            ROBOT.MoveJ(joints)
        except Exception as e:
            if DEBUG:
                print(f"Error moving to configuration: {e}")
                debuglist.append(f"Error moving to configuration: {e}")
            continue  # Skip this configuration

        # Check for collisions without moving
        try:
            RDK.setCollisionActive(COLLISION_ON)
            collision = RDK.Collisions()

            # If no collision, we found a valid configuration
            if collision == 0:
                return 0

        except Exception as e:
            if DEBUG:
                print(f"Error checking collision: {e}")
                debuglist.append(f"Error checking collision: {e}")
            continue  # Skip this configuration on error

    # All configurations had issues
    return 1

def test_collision_target(target):
    """
    Test if the current target pose is collision-free.
    Optimized to quickly check multiple configurations.
    """
    try:
        if DEBUG:
            print("Testing target for collisions")
            debuglist.append("Testing target for collisions")

        # Get all possible configurations for this target
        possible_configurations = ROBOT.SolveIK_All(target.Pose(), tool=TOOLPOSE, reference=FRAMEPOSE)

        # Quick check - if no configurations are possible, fail early
        if not possible_configurations or len(possible_configurations) == 0:
            return -2

        # Test configurations in batches for efficiency
        return test_all_configurations(possible_configurations)

    except Exception as e:
        if DEBUG:
            print(f"Error in test_collision_target: {e}")
            debuglist.append(f"Error in test_collision_target: {e}")
        return 1  # Assume collision on error

def test_issues_point(target, rz):
    if DEBUG:
        print("testing point")
        debuglist.append("testing point")

    # define the rotated position to test for collisions
    target_new_pose = RelTool(target.Pose(), 0,0,0, 0,0,rz)
    possible_robot_configurations = ROBOT.SolveIK_All(target_new_pose, tool=TOOLPOSE, reference=FRAMEPOSE)
    issues_value = test_all_configurations(possible_robot_configurations) # returns 0 if at least one configuration is without issues

    return issues_value, target_new_pose

rotation_direction = "pos"
direction_changes = 0
holes_no_solution = []

def find_collision_free_configuration(target, idx):
    """
    Find a collision-free configuration for the target by trying different rotations.
    This version avoids script interruption on collision detection.

    Returns:
        True if a collision-free configuration was found, False otherwise
    """
    # Store original pose to restore if needed
    original_pose = target.Pose()

    # First check if original pose is collision-free
    result = test_collision_safe(original_pose)
    if result == 0:
        if DEBUG:
            print(f"Original pose for Hole {idx} is collision-free")
            debuglist.append(f"Original pose for Hole {idx} is collision-free")
        return True

    # Define rotation search strategy
    # Use an incremental approach rather than testing all at once
    rotation_axes = ['z', 'y', 'x']  # Order matters - most likely axis first
    angles_to_try = [15, 30, 45, 60, 90, 120, 150, 180, -15, -30, -45, -60, -90, -120, -150, -180]

    # Track best rotation setup
    best_result = 1  # 1 = collision, we want 0 = no collision
    best_pose = None

    # Try each axis and angle combination
    for axis in rotation_axes:
        for angle in angles_to_try:
            try:
                # Create a new rotated pose
                if axis == 'z':
                    new_pose = RelTool(original_pose, 0, 0, 0, 0, 0, angle)
                elif axis == 'y':
                    new_pose = RelTool(original_pose, 0, 0, 0, 0, angle, 0)
                elif axis == 'x':
                    new_pose = RelTool(original_pose, 0, 0, 0, angle, 0, 0)

                # Test this pose
                result = test_collision_safe(new_pose)

                # If collision-free, we can use this one
                if result == 0:
                    if DEBUG:
                        print(f"Found collision-free pose for Hole {idx} with {axis} rotation of {angle}")
                        debuglist.append(f"Found collision-free pose for Hole {idx} with {axis} rotation of {angle}")

                    # Set the target pose and return success
                    target.setPose(new_pose)
                    return True

                # Update best result if this is better
                if result < best_result:
                    best_result = result
                    best_pose = new_pose

            except Exception as e:
                if DEBUG:
                    print(f"Error testing {axis} rotation of {angle} for Hole {idx}: {e}")
                    debuglist.append(f"Error testing {axis} rotation of {angle} for Hole {idx}: {e}")

    # If we get here, no completely collision-free pose was found
    # If we found a feasible but colliding pose, use that as a fallback
    if best_pose is not None:
        try:
            target.setPose(best_pose)
            if DEBUG:
                print(f"Using best available pose for Hole {idx} (not collision-free)")
                debuglist.append(f"Using best available pose for Hole {idx} (not collision-free)")
        except:
            # If setting pose fails, restore original
            target.setPose(original_pose)
    else:
        # Restore original pose
        target.setPose(original_pose)

    if DEBUG:
        print(f"No collision-free pose found for Hole {idx}")
        debuglist.append(f"No collision-free pose found for Hole {idx}")

    return False

def rotate_target(pose, axis, angle):
    """Rotate target pose around specified axis by given angle."""
    try:
        if axis.lower() == 'z':
            return RelTool(pose, 0, 0, 0, 0, 0, angle)
        elif axis.lower() == 'y':
            return RelTool(pose, 0, 0, 0, 0, angle, 0)
        elif axis.lower() == 'x':
            return RelTool(pose, 0, 0, 0, angle, 0, 0)
        else:
            return pose
    except Exception as e:
        if DEBUG:
            print(f"Error rotating target ({axis}, {angle}): {e}")
            debuglist.append(f"Error rotating target ({axis}, {angle}): {e}")
        return pose



def main():
    global holes_no_solution
    holes_no_solution = []

    MAKE_GUI_PROGRAM = True

    ROBOT.setFrame(FRAME)
    ROBOT.setTool(TOOL)

    if RDK.RunMode() == RUNMODE_SIMULATE:
        MAKE_GUI_PROGRAM = True
    else:
        MAKE_GUI_PROGRAM = False

    if MAKE_GUI_PROGRAM:
        # Disable rendering for speed
        RDK.Render(False)

        # Process the targets
        holes_no_solution = make_targets(csv_file)

        # Re-enable rendering
        RDK.Render(True)

        # Final report
        if holes_no_solution:
            final_message = f"Completed with {len(holes_no_solution)} holes without solution: {holes_no_solution}"
            RDK.ShowMessage(final_message, False)
            if DEBUG:
                print(final_message)
                debuglist.append(final_message)

                # Write debug info to file
                current_time = datetime.datetime.now()
                filename = os.path.splitext(os.path.basename(__file__))
                with open("debugfile.txt", "a") as file:
                    file.write("\n\n-----------------------------------------------\n")
                    file.write(current_time.strftime("%c"))
                    file.write("\n-----------------------------------------------\n")
                    for prints in debuglist:
                        file.write(str(prints))
                        file.write("\n")
                    file.write(str(holes_no_solution))
                    file.write(str(filename[0]))

# Run the main function
if __name__ == "__main__":
    main()
else:
    main()  # For RoboDK compatibility, run even if imported

--- Python program csv_importernewest ---
# This macro can load CSV files from Denso programs in RoboDK.
# Supported types of files are:
#  1-Tool data : Tool.csv
#  2-Work object data: Work.csv
#  3-Target data: P_Var.csv
# This macro can also filter a given targets file

# Type help("robodk.robolink") or help("robodk.robomath") for more information
# Press F5 to run the script
# Visit: http://www.robodk.com/doc/PythonAPI/
# For RoboDK API documentation

import os
import datetime

import tkinter as tk
from tkinter import messagebox

from robodk.robolink import *  # API to communicate with RoboDK
from robodk.robomath import *  # Robot toolbox
from robodk.robodialogs import *
from robodk.robofileio import *
import robodk.robolinkutils as RDKutils

DEBUG = False

debuglist = []

# Start communication with RoboDK
RDK = Robolink()

# Ask the user to select the robot
ROBOT = RDK.ItemUserPick('Select a robot', ITEM_TYPE_ROBOT)

# Check if the user selected a robot
if not ROBOT.Valid():
    quit()


# Ask the user to select a reference frame and get the active tool
BASE = ROBOT.Parent()
#BASE = RDK.Item('UR10e Base', ITEM_TYPE_FRAME)
#BASE = RDK.ItemUserPick('Select robot base frame', ITEM_TYPE_FRAME)
FRAME = RDK.ItemUserPick('Reference Frame', ITEM_TYPE_FRAME)
FRAMEPOSE = RDKutils.getPoseWrt(FRAME, BASE) #frame pose wrt robot base
TOOL = ROBOT.getLink(ITEM_TYPE_TOOL)
TOOLPOSE = RDKutils.getPoseWrt(TOOL, TOOL.Parent()) #tool pose wrt robot flange

if not FRAME.Valid() or not TOOL.Valid():
    raise Exception("Select appropriate FRAME and TOOL references")


# Function to convert XYZWPR to a pose
# Important! Specify the order of rotation
def xyzwpr_to_pose(xyzwpr):
    x, y, z, rx, ry, rz = xyzwpr
    return point_Zaxis_2_pose([x, y, z], [-rx, -ry, -rz])
    #return transl(x, y, z) * rotz(rz * pi / 180) * roty(ry * pi / 180) * rotx(rx * pi / 180)
    #return transl(x,y,z)*rotx(rx*pi/180)*roty(ry*pi/180)*rotz(rz*pi/180)
    #return KUKA_2_Pose(xyzwpr)


# csv_file = 'C:/Users/Albert/Desktop/Var_P.csv'
csv_file = getOpenFileName(RDK.getParam('PATH_OPENSTATION'))

# Specify file codec
codec = 'utf-8'  #'ISO-8859-1'


# Load P_Var.CSV data as a list of poses, including links to reference and tool frames
def load_targets(strfile):
    csvdata = LoadList(strfile, ',', codec)
    poses = []
    idxs = []
    for i in range(0, len(csvdata)):
        x, y, z, rx, ry, rz = csvdata[i][0:6]
        poses.append(xyzwpr_to_pose([x, y, z, rx, ry, rz]))
        #idxs.append(csvdata[i][6])
        idxs.append(i)

    return poses, idxs


# Load and display Targets from P_Var.CSV in RoboDK
def make_targets(strfile):
    poses, idxs = load_targets(strfile)
    program_name = getFileName(strfile)
    program_name = program_name.replace('-', '_').replace(' ', '_')

    for pose, idx in zip(poses, idxs):
        name = 'H-%s-%i' % (program_name, idx)
        target = RDK.Item(name, ITEM_TYPE_TARGET)
        if target.Valid():
            target.Delete()
        target = RDK.AddTarget(name, FRAME, ROBOT)


        target.setPose(pose)
        collision_free(target, idx)

def test_all_configurations(configurations):
    for joints in configurations:

        # turn collision checking off
        RDK.setCollisionActive(COLLISION_OFF)
        if DEBUG:
            is_active = RDK.Command("CollisionActive")
            print(f"collsion active? should be off (0) {is_active}")
            debuglist.append(f"collsion active? should be off (0) {is_active}")

        # move to target
        try:
            ROBOT.MoveJ(joints)
        except TargetReachError:
            continue

        # turn collision checking on, test for collisions
        RDK.setCollisionActive(COLLISION_ON)
        if DEBUG:
            is_active = RDK.Command("CollisionActive")
            print(f"collsion active? should be on (1) {is_active}")
            debuglist.append(f"collsion active? should be on (1) {is_active}")

        collision = RDK.Collisions()
        if DEBUG:
            print(f"collision: {collision}")
            debuglist.append(f"collision: {collision}")

        collision_items = RDK.CollisionItems()
        if TOOL in collision_items or collision == 0:
            break

    try:
        collision
    except NameError:
        collision = -2
        if DEBUG:
            print("Target cannot be reached or is to close to a singularity")
            debuglist.append("Target cannot be reached or is to close to a singularity")

    return collision


def test_collision_target(target, rz):
    if DEBUG:
        print("testing at target")
        debuglist.append("testing at target")

    possible_robot_configurations = ROBOT.SolveIK_All(target.Pose(), tool=TOOLPOSE, reference=FRAMEPOSE)
    issues_value = test_all_configurations(possible_robot_configurations) # returns 0 if at least one configuration is without issues

    return issues_value

def test_issues_point(target, rz, flip_approach=False):
    if DEBUG:
        print("testing point")
        debuglist.append("testing point")

    # Get the original pose
    original_pose = target.Pose()

    # For vertical walls, we might need to completely flip the approach
    if flip_approach:
        # Rotate 180 degrees around Y axis (assuming Y is the axis parallel to the wall)
        # This effectively approaches from the opposite direction
        target_new_pose = RelTool(original_pose, 0, 0, 0, 0, 180, 0)
        # Then apply the requested Z rotation
        target_new_pose = RelTool(target_new_pose, 0, 0, 0, 0, 0, rz)
    else:
        # Standard rotation around Z axis only
        target_new_pose = RelTool(original_pose, 0, 0, 0, 0, 0, rz)

    possible_robot_configurations = ROBOT.SolveIK_All(target_new_pose, tool=TOOLPOSE, reference=FRAMEPOSE)
    issues_value = test_all_configurations(possible_robot_configurations)

    return issues_value, target_new_pose

rotation_direction = "pos"
direction_changes = 0
holes_no_solution = []

def collision_free(target, idx):
    rotation_step = 10
    repmax = 360/rotation_step
    global rotation_direction
    global direction_changes
    s = 0
    rep = 0

    if DEBUG:
        print(f"\nHole {idx}")
        debuglist.append(f"\nHole {idx}")

    # First try the original approach
    issues_value, target_new_pose = test_issues_point(target, 0, flip_approach=False)

    # If there's a collision, try different approaches
    while issues_value != 0 and s < 100:
        if DEBUG:
            print(f"s before: {s}")
            debuglist.append(f"s before: {s}")
            print(f"rep: {rep}")
            debuglist.append(f"rep: {rep}")
            print(f"rotation direction: {rotation_direction}")
            debuglist.append(f"rotation direction: {rotation_direction}")
            print(f"direction changes: {direction_changes}")
            debuglist.append(f"direction changes: {direction_changes}")

        s += 1

        # For unreachable targets or potential vertical wall collision situations
        if issues_value == -2 and direction_changes < 2:
            if rotation_direction == "pos":
                rotation_direction = "neg"
                direction_changes += 1
                r = -1
            else:
                rotation_direction = "pos"
                direction_changes += 1
                r = 1

            # Try the opposite approach direction if we've changed direction once already
            # This is key for vertical walls
            if direction_changes >= 1:
                issues_value, target_new_pose = test_issues_point(target, r*rotation_step, flip_approach=True)
            else:
                issues_value, target_new_pose = test_issues_point(target, r*rotation_step, flip_approach=False)

            target.setPose(target_new_pose)

        # For collision situations, rotate around Z
        elif issues_value > 0 and rep < repmax:
            RDK.setCollisionActive(COLLISION_OFF)
            if DEBUG:
                is_active = RDK.Command("CollisionActive")
                print(f"collsion active? should be off (0) {is_active}")
                debuglist.append(f"collsion active? should be off (0) {is_active}")

            ROBOT.MoveJ(target.Pose())

            if rotation_direction == "neg":
                r = -1
            elif rotation_direction == "pos":
                r = 1

            # After trying several rotations, try the flip approach
            if rep > repmax/2:
                issues_value, target_new_pose = test_issues_point(target, r*rotation_step, flip_approach=True)
            else:
                issues_value, target_new_pose = test_issues_point(target, r*rotation_step, flip_approach=False)

            target.setPose(target_new_pose)
            rep += 1

        elif direction_changes >= 2 or rep >= repmax:
            break

        else:
            RDK.ShowMessage(f"Unknown error occured at Hole {idx} while looking for collision free position")
            if DEBUG:
                print(f"Unknown error occured at Hole {idx} while looking for collision free position")
                debuglist.append(f"Unknown error occured at Hole {idx} while looking for collision free position")

    direction_changes = 0
    if issues_value == 0:
        print(f"No issues at Hole {idx}")
        debuglist.append(f"No issues at Hole {idx}")
    elif direction_changes >= 2 or rep >= repmax or s >= 100:
        RDK.ShowMessage(f"No solution found for Hole {idx}", False)
        holes_no_solution.append(idx)
        if DEBUG:
            print(f"No solution found for Hole {idx}")
            debuglist.append(f"No solution found for Hole {idx}")
    else:
        RDK.ShowMessage(f"Unknown error occured at Hole {idx} while looking for collision free position")
        if DEBUG:
            print(f"Unknown error occured at Hole {idx} while looking for collision free position")
            debuglist.append(f"Unknown error occured at Hole {idx} while looking for collision free position")


MAKE_GUI_PROGRAM = True

ROBOT.setFrame(FRAME)
ROBOT.setTool(TOOL)

if RDK.RunMode() == RUNMODE_SIMULATE:
    MAKE_GUI_PROGRAM = True
    # MAKE_GUI_PROGRAM = mbox('Do you want to create a new program? If not, the robot will just move along the targets', 'Yes', 'No')
else:
    # if we run in program generation mode just move the robot
    MAKE_GUI_PROGRAM = False

if MAKE_GUI_PROGRAM:
    RDK.Render(False)  # Faster if we turn render off
    make_targets(csv_file)
else:
    l

if len(holes_no_solution) != 0:
    RDK.ShowMessage(f"Holes without solution: {holes_no_solution}")

if DEBUG:
    print(f"Holes without solution: {holes_no_solution}")
    debuglist.append(f"Holes without solution: {holes_no_solution}")

    current_time = datetime.datetime.now()
    filename = os.path.splitext(os.path.basename(__file__))
    with open("C:/Users/Laura/Documents/1.Windesheim/Stage/2024/Lectoraat/Deelvragen/2.Targets maken/debugfile.txt", "a") as file:
        file.write("\n\n-----------------------------------------------\n")
        file.write(current_time.strftime("%c"))
        file.write("\n-----------------------------------------------\n")
        for prints in debuglist:
            file.write(prints)
            file.write("\n")
        file.write(holes_no_solution)
        file.write(filename[0])

--- Python program Make_approaches_paths ---
from robodk.robolink import *  # API to communicate with RoboDK
from robodk.robomath import *  # Robot toolbox
import robodk.robolinkutils as RDKutils


DEBUG = False


# Link to RoboDK
RDK = Robolink()

ROBOT = RDK.ItemUserPick('Select a Robot', ITEM_TYPE_ROBOT)
FRAME = RDK.ItemUserPick('Reference Frame', ITEM_TYPE_FRAME)

if not ROBOT.Valid() or not FRAME.Valid():
    raise Exception("Select appropriate ROBOT and FRAME")

BASE = RDK.Item('UR10e Base', ITEM_TYPE_FRAME)
#BASE = RDK.ItemUserPick('Select robot base frame', ITEM_TYPE_FRAME)
FRAMEPOSE = RDKutils.getPoseWrt(FRAME, BASE) #frame pose wrt robot base
TOOL = ROBOT.getLink(ITEM_TYPE_TOOL)
TOOLPOSE = RDKutils.getPoseWrt(TOOL, TOOL.Parent()) #tool pose wrt robot flange




# get all the holes as items
All_items = RDK.ItemList(ITEM_TYPE_TARGET)
#RDK_items = [item for item in All_items if "Hole" in item.Name()]
RDK_items = [item for item in All_items if "H" in item.Name()]
print(f"Holes: {len(RDK_items)}")

RDK.setCollisionActive(COLLISION_OFF)

def print_xyzrpw(pose):
    x, y, z, rx, ry, rz = pose_2_xyzrpw(pose)
    print(x, y, z, rx, ry, rz)


class Hole:
    def __init__(self, pose, target):
        self.pose = pose
        self.target = target
        self.name = self.target.Name()
        self.split_position_rotation(pose)

    def split_position_rotation(self, pose):
        x, y, z, rx, ry, rz = pose_2_xyzrpw(pose)
        self.position = x, y, z
        # get the way the z-axis is facing
        self.rotation = pose[0:3,2] # from all 3 rows (0:3) only the 3rd column (index 2) (the last column of the rotation matrix)
        # format the z-axis facing, so it can be made a key in the dictonary
        zfacing1 = round(self.rotation.tolist()[0])
        zfacing2 = round(self.rotation.tolist()[1])
        zfacing3 = round(self.rotation.tolist()[2])
        self.rot_identifier = f"{zfacing1}_{zfacing2}_{zfacing3}"

class Face:
    def __init__(self, key):
        self.key = key
        self.get_midpoint(key)
        self.rotation = self.holes[0].rotation.tolist()
        self.offset_multiplier = self.rotation
        self.approaches = []

    def get_midpoint(self, key):
        #global dic
        #targets from key
        self.holes = dic[key]
        #x, y, z from targets
        self.x_values = []
        self.y_values = []
        self.z_values = []
        for hole in self.holes:
            x, y, z = hole.position
            self.x_values.append(x)
            self.y_values.append(y)
            self.z_values.append(z)
        if DEBUG:
            print("ranges:")
            print(self.x_values)
            print(self.y_values)
            print(self.z_values)
        #min and max of these
        self.x_values.sort()
        min_x = self.x_values[0]
        max_x = self.x_values[len(self.x_values)-1]
        offset_x = (max_x - min_x)/2
        mid_x = max_x - offset_x
        self.xranges = min_x, max_x, mid_x

        self.y_values.sort()
        min_y = self.y_values[0]
        max_y = self.y_values[len(self.y_values)-1]
        offset_y = (max_y - min_y)/2
        mid_y = max_y - offset_y
        self.yranges = min_y, max_y, mid_y

        self.z_values.sort()
        min_z = self.z_values[0]
        max_z = self.z_values[len(self.z_values)-1]
        offset_z = (max_z - min_z)/2
        mid_z = max_z - offset_z
        self.zranges = min_z, max_z, mid_z

        self.midpoint = mid_x, mid_y, mid_z

        self.ref_hole = self.holes[0]
        ref_pose = self.ref_hole.pose
        ref_pose[0,3] = mid_x
        ref_pose[1,3] = mid_y
        ref_pose[2,3] = mid_z
        self.midpose = ref_pose
        if DEBUG:
            print("min, max, mid: ")
            print("x: ", self.xranges)
            print("y: ", self.yranges)
            print("z: ", self.zranges)
            print("midpoint: ", self.midpoint)
            print("midpose: ", self.midpose)

    def add_approaches(self, approach):
        self.approaches.append(approach)



class Approach:
    def __init__(self, face, number):
        self.face = face
        self.number = number
        self.target = self.make_approach_target(face, number)

    def make_approach_target(self, face, number):
        approach_point = self.get_approach_point(face)
        approach_target = RDK.Item(f"approach {idx} {face.rotation}", ITEM_TYPE_TARGET)
        if approach_target.Valid():
            approach_target.Delete()
        approach_target = RDK.AddTarget(f"approach {idx} {face.rotation}", FRAME, ROBOT)
        approach_target.setPose(approach_point)
        if DEBUG:
            print("approach target:\n", approach_point)
        return approach_target

    def get_approach_point(self, face):
        MAX_APPROACH = 100 #in mm
        MIN_APPROACH = 20 #in mm
        STEP = 40 #in mm
        ROT_STEP = 20 #in degrees
        approach_point = self.test_distance(face, MAX_APPROACH, MIN_APPROACH, STEP, ROT_STEP)
        return approach_point

    def test_distance(self, face, MAX_APPROACH, MIN_APPROACH, STEP, ROT_STEP):
        approach_distance = MAX_APPROACH
        rep = 0
        repmax = 360/ROT_STEP
        rot_offset = 0
        rotation_direction = "pos"
        direction_changes = 0

        z = approach_distance
        issues, approach_point = self.test_point(face.midpose, z, 0)
        #first_issues_value = issues
        if issues == -2:
            rz = 180
            rot_offset = rz
            issues, approach_point = self.test_point(face.midpose, z, rz)

        sa = 0
        while issues != 0 and approach_distance >= MIN_APPROACH + STEP and sa < 100:
            sa += 1
            approach_distance -= STEP
            z = approach_distance
            rz = 0
            issues, approach_point = self.test_point(face.midpose, z, rz)
            issues, approach_point = self.rotate(face, issues, approach_distance, rot_offset, ROT_STEP)

        return approach_point

    def rotate(self, face, issues, approach_distance, rot_offset, ROT_STEP):
        repmax = 360/ROT_STEP
        rotation_direction = "pos"
        direction_changes = 0
        rep = 0
        sb = 0
        while issues != 0 and sb < 100:
            sb += 1
            if issues == -2 and direction_changes < 2:
                if rotation_direction == "pos":
                    rotation_direction = "neg"
                    r = -1 #rotation factor to make the rotation negative
                else:
                    rotation_direction = "pos"
                    r = 1
                direction_changes += 1
                z = approach_distance
                rz = rot_offset + r * ROT_STEP
                issues, approach_point = self.test_point(face.midpose, z, rz)
            elif issues > 0 and rep < repmax:
                if rotation_direction == "neg":
                    r = -1
                else:
                    r = 1
                rep += 1
                z = approach_distance
                rz = rot_offset + r * ROT_STEP
                rot_offset = rz
                issues, approach_point = self.test_point(face.midpose, z, rz)
            elif direction_changes >= 2 or rep >= repmax:
                break

            else:
                print(f"Unknown error occured at Approach {self.number}")

        if issues != 0 and (direction_changes >= 2 or rep >= repmax or sb == 100):
            print(f"No solution found for Approach {self.number}")
            global approach_noSolution
            approach_noSolution.append(self.number)
            RDK.ShowMessage(f"No solution found for Approach {self.number}", False)
        return issues, approach_point

    def test_point(self, point, z, rz):
        # define the position to test for collisions
        test_point = RelTool(point, 0,0,z, 0,0,rz)
        possible_robot_configurations = ROBOT.SolveIK_All(test_point, tool=TOOLPOSE, reference=FRAMEPOSE)
        issues = self.test_all_configurations(possible_robot_configurations)
        return issues, test_point

    def test_all_configurations(self, configurations):
        for joints in configurations:

            # turn collision checking off
            RDK.setCollisionActive(COLLISION_OFF)
            is_active = RDK.Command("CollisionActive")
            #print(f"collsion active? should be off (0) {is_active}")

            # move to target
            try:
                ROBOT.MoveJ(joints)
            except TargetReachError:
                continue

            # turn collision checking on, test for collisions
            RDK.setCollisionActive(COLLISION_ON)
            is_active = RDK.Command("CollisionActive")
            #print(f"collsion active? should be on (1) {is_active}")
            collision = RDK.Collisions()
            #print(f"collision: {collision}")
            collision_items = RDK.CollisionItems()
            if TOOL in collision_items or collision == 0:
                break

        try:
            collision
        except NameError:
            collision = -2 # TargetReachError occures for every configuration
            #print("Target cannot be reached or is to close to a singularity")

        return collision

def collision_free_paths(face, approach):
    possible_configurations = ROBOT.SolveIK_All(approach.target.Pose(), tool=TOOLPOSE, reference=FRAMEPOSE)
    for i, joints in enumerate(possible_configurations):
        print(f"testing configuration {i+1}")
        for j, hole in enumerate(face.holes):
            RDK.setCollisionActive(COLLISION_OFF)
            ROBOT.MoveJ(joints)
            RDK.setCollisionActive(COLLISION_ON)
            issues = ROBOT.MoveJ_Test(joints, hole.target.Joints())
            print(f"Hole {hole.name} with issues = {issues}")
            if issues == 0:
                continue
            break

        if issues == 0:
            print(f"found valid configuration: {i+1}")
            approach.target.setJoints(joints)
            break

    if issues != 0:
        print(f"no configuration found for approach {approach.number}")
        path_no_solution.append(hole.name)

holes = []
dic = {}
faces = []
approach_noSolution = []
path_no_solution = []

# convert the target items into target objects
for item in RDK_items:
    hole = Hole(item.Pose(), item)
    holes.append(hole)

# put the targets with the z-axis facing the same way together
for hole in holes:
    if hole.rot_identifier in dic:
        #dic exists put it in
        dic[hole.rot_identifier].append(hole)
    else:
        #make a dic and put it in
        dic[hole.rot_identifier] = [hole]

keys = list(dic.keys())
for key in keys:
    if DEBUG:
        print(f"{key}: {dic[key]}")
    face = Face(key)
    faces.append(face)
    if DEBUG:
        print(face.midpoint)

for idx, face in enumerate(faces):
    if DEBUG:
        print(faces)
    approach = Approach(face, idx)
    face.add_approaches(approach)

    #paden maken tussen approach en targets die daar bij horen
    for approach in face.approaches:
        collision_free_paths(face, approach)
        for hole in face.holes:
            program_name = f"to {hole.name}"
            program = RDK.Item(program_name, ITEM_TYPE_PROGRAM)
            if program.Valid():
                program.Delete()
            program = RDK.AddProgram(program_name, ROBOT)
            ROBOT.MoveJ(approach.target)
            program.MoveJ(hole.target)

--- Python program TargetFixer ---
from robodk import robolink, robomath
import robodk.robolinkutils as RDKutils

from robodk.robolink import *       # RoboDK API
from robodk.robomath import *        # Math toolbox (provides transl, etc.)
from robodk.robodialogs import *
from robodk.robofileio import *

def main():
    # Initialize RoboDK instance
    RDK = robolink.Robolink()

    # Let the user pick a Robot and a Reference Frame
    ROBOT = RDK.ItemUserPick('Select a Robot', ITEM_TYPE_ROBOT)
    FRAME = RDK.ItemUserPick('Select a Reference Frame', ITEM_TYPE_FRAME)
    if not ROBOT.Valid() or not FRAME.Valid():
        raise Exception("Select appropriate ROBOT and FRAME")

    # Get Base, Tool and FRAME pose (adjust names as needed)
    BASE = RDK.Item('UR10e Base', ITEM_TYPE_FRAME)
    FRAMEPOSE = RDKutils.getPoseWrt(FRAME, BASE) if BASE.Valid() else FRAME.Pose()
    TOOL = ROBOT.getLink(ITEM_TYPE_TOOL)
    TOOLPOSE = RDKutils.getPoseWrt(TOOL, TOOL.Parent())

    # Activate collision checking
    RDK.setCollisionActive(COLLISION_ON)

    # Get all targets (or filter them as needed)
    all_targets = RDK.ItemList(ITEM_TYPE_TARGET)

    fixed_targets = []
    unfixed_targets = []

    # Process every target one by one
    for target in all_targets:
        original_pose = target.Pose()
        print(f"\nProcessing target: {target.Name()}")

        # First, check if the target is already collision free:
        if not target_in_collision(RDK, ROBOT, target, FRAMEPOSE, TOOLPOSE):
            print(f"Target {target.Name()} is already collision free. No fix needed.")
            continue

        print(f"Target {target.Name()} is in collision. Attempting to fix by shifting along principal axes...")

        # Try to fix by shifting along X, then Y, then Z
        fixed = fix_target(target, original_pose, RDK, ROBOT, FRAMEPOSE, TOOLPOSE)
        if fixed:
            fixed_targets.append(target.Name())
        else:
            unfixed_targets.append(target.Name())
            target.setPose(original_pose)  # revert to original if no fix was found

    # Summary report
    print("\nTarget fixing complete.")
    print("Fixed targets:")
    for t in fixed_targets:
        print("  -", t)
    if unfixed_targets:
        print("Targets that could not be fixed:")
        for t in unfixed_targets:
            print("  -", t)

def target_in_collision(RDK, ROBOT, target, FRAMEPOSE, TOOLPOSE):
    """
    Checks whether the given target causes a collision.
    It does so by attempting to solve IK and simulating a MoveJ.
    Returns True if a collision (or no valid configuration) is detected.
    """
    pose = target.Pose()
    possible_configs = ROBOT.SolveIK_All(pose, tool=TOOLPOSE, reference=FRAMEPOSE)
    if not possible_configs:
        return True
    for joints in possible_configs:
        try:
            ROBOT.MoveJ(joints)
        except Exception:
            continue
        if not RDK.Collisions():
            return False
    return True

def fix_target(target, original_pose, RDK, ROBOT, FRAMEPOSE, TOOLPOSE):
    """
    Attempts to fix a target by shifting it along each principal axis.

    For each axis (X, Y, Z), the function:
      - Tries a positive shift in 10-mm increments (10 steps).
      - Reverts to the original pose.
      - Tries a negative shift in 10-mm increments (10 steps).

    If a collision-free pose is found during any of these tests, the target is updated.
    Returns True if a valid pose is found, otherwise False.
    """
    # Define axes along which to shift using lambda functions that generate translation matrices.
    # The transl(x, y, z) function creates a translation matrix in the local coordinate system when multiplied with a pose.
    axes = [
        ("X", lambda d: transl(d, 0, 0)),
        ("Y", lambda d: transl(0, d, 0)),
        ("Z", lambda d: transl(0, 0, d))
    ]

    # For each axis...
    for axis_name, shift_func in axes:
        # Try positive direction shifts first
        for i in range(1, 11):
            shift_matrix = shift_func(10 * i)  # 10-mm increments
            test_pose = original_pose * shift_matrix
            target.setPose(test_pose)
            if not target_in_collision(RDK, ROBOT, target, FRAMEPOSE, TOOLPOSE):
                print(f"Target {target.Name()} fixed with a +{10*i} mm shift along {axis_name}.")
                return True
        # Revert to the original pose before trying the negative direction
        target.setPose(original_pose)
        for i in range(1, 11):
            shift_matrix = shift_func(-10 * i)
            test_pose = original_pose * shift_matrix
            target.setPose(test_pose)
            if not target_in_collision(RDK, ROBOT, target, FRAMEPOSE, TOOLPOSE):
                print(f"Target {target.Name()} fixed with a {-10*i} mm shift along {axis_name}.")
                return True
        # Revert to the original pose before trying the next axis
        target.setPose(original_pose)
    return False

if __name__ == '__main__':
    main()

--- Python program generatefaceapproaches ---
from robodk.robolink import *  # API to communicate with RoboDK
from robodk.robomath import *   # Robot toolbox
import robodk.robolinkutils as RDKutils
from robodk import robolink

DEBUG = False

# Link to RoboDK
RDK = Robolink()

ROBOT = RDK.ItemUserPick('Select a Robot', ITEM_TYPE_ROBOT)
FRAME = RDK.ItemUserPick('Reference Frame', ITEM_TYPE_FRAME)

if not ROBOT.Valid() or not FRAME.Valid():
    raise Exception("Select appropriate ROBOT and FRAME")

BASE = RDK.Item('UR10e Base', ITEM_TYPE_FRAME)
FRAMEPOSE = RDKutils.getPoseWrt(FRAME, BASE)  # frame pose with respect to robot base
TOOL = ROBOT.getLink(ITEM_TYPE_TOOL)
TOOLPOSE = RDKutils.getPoseWrt(TOOL, TOOL.Parent())  # tool pose with respect to robot flange

# Get all the holes as targets (only those with "H" in the name)
All_items = RDK.ItemList(ITEM_TYPE_TARGET)
RDK_items = [item for item in All_items if "H" in item.Name()]
print(f"Holes: {len(RDK_items)}")

RDK.setCollisionActive(COLLISION_OFF)

def print_xyzrpw(pose):
    x, y, z, rx, ry, rz = pose_2_xyzrpw(pose)
    print(x, y, z, rx, ry, rz)

class Hole:
    def __init__(self, pose, target):
        self.pose = pose
        self.target = target
        self.name = self.target.Name()
        self.split_position_rotation(pose)

    def split_position_rotation(self, pose):
        x, y, z, rx, ry, rz = pose_2_xyzrpw(pose)
        self.position = (x, y, z)
        # Get the z-axis direction (3rd column of the rotation matrix)
        self.rotation = pose[0:3, 2]
        zfacing1 = round(self.rotation.tolist()[0])
        zfacing2 = round(self.rotation.tolist()[1])
        zfacing3 = round(self.rotation.tolist()[2])
        self.rot_identifier = f"{zfacing1}_{zfacing2}_{zfacing3}"

class Face:
    def __init__(self, key):
        self.key = key
        self.get_midpoint(key)
        self.rotation = self.holes[0].rotation.tolist()
        self.offset_multiplier = self.rotation
        self.approaches = []  # Not used in the new functions

    def get_midpoint(self, key):
        # Retrieve all holes corresponding to this face
        self.holes = dic[key]
        x_values = [hole.position[0] for hole in self.holes]
        y_values = [hole.position[1] for hole in self.holes]
        z_values = [hole.position[2] for hole in self.holes]

        # Sort and compute the midpoint as the average of the min and max values
        x_values.sort()
        y_values.sort()
        z_values.sort()
        min_x, max_x = x_values[0], x_values[-1]
        min_y, max_y = y_values[0], y_values[-1]
        min_z, max_z = z_values[0], z_values[-1]

        mid_x = (min_x + max_x) / 2
        mid_y = (min_y + max_y) / 2
        mid_z = (min_z + max_z) / 2

        self.midpoint = (mid_x, mid_y, mid_z)

        # Use the first hole's pose as a template and update its translation to the midpoint
        self.ref_hole = self.holes[0]
        ref_pose = self.ref_hole.pose
        ref_pose[0, 3] = mid_x
        ref_pose[1, 3] = mid_y
        ref_pose[2, 3] = mid_z
        self.midpose = ref_pose

    def add_approaches(self, approach):
        self.approaches.append(approach)

# --- Process holes and group them into faces based on z-axis orientation ---
holes = []
dic = {}
faces = []

# Convert the target items into Hole objects
for item in RDK_items:
    hole = Hole(item.Pose(), item)
    holes.append(hole)

# Group holes with the same z-axis orientation (rounded)
for hole in holes:
    if hole.rot_identifier in dic:
        dic[hole.rot_identifier].append(hole)
    else:
        dic[hole.rot_identifier] = [hole]

# Create Face objects from the groups
for key in dic:
    face = Face(key)
    faces.append(face)

# --- NEW FUNCTION: Create face targets at the midpoint of each face ---
def create_face_targets():
    """
    For each computed face, create a new target in RoboDK at the face midpoint.
    """
    for face in faces:
        face_target_name = f"Face_Target_{face.key}"
        existing_target = RDK.Item(face_target_name, ITEM_TYPE_TARGET)
        if existing_target.Valid():
            existing_target.Delete()
        face_target = RDK.AddTarget(face_target_name, FRAME, ROBOT)
        # face_target.setAsJointTarget() # joint target ?
        # face_target.setJoints(ROBOT.Joints())
        face_target.setPose(face.midpose)
        print(f"Created face target for face {face.key} at midpoint {face.midpoint}")

# --- NEW FUNCTION: Create a program for each face using MoveL commands ---
def create_face_programs():
    """
    For each face, generate a program that moves from the face target (approach target)
    to every hole target on that face using a MoveL command.
    Each move from the face target to a hole target is followed by a return move to the face target.
    """
    for face in faces:
        face_target_name = f"Face_Target_{face.key}"
        face_target = RDK.Item(face_target_name, ITEM_TYPE_TARGET)
        prog_name = f"Program_Face_{face.key}"
        existing_prog = RDK.Item(prog_name, ITEM_TYPE_PROGRAM)
        if existing_prog.Valid():
            existing_prog.Delete()
        prog = RDK.AddProgram(prog_name, ROBOT)

        # Add a move to the face target as the starting (approach) move
        prog.MoveL(face_target)

        # For each hole in this face, add a MoveL to go to the hole target and then a MoveL back to the face target.
        for hole in face.holes:
            prog.MoveL(hole.target)
            # prog.RunInstruction('move_shank(20)', robolink.INSTRUCTION_CALL_PROGRAM)  # Tighten screw
            # prog.RunInstruction('move_shank(0)', robolink.INSTRUCTION_CALL_PROGRAM)  # Release screwdriver


            prog.MoveL(face_target)
            print(f"Program {prog_name}: Added MoveL from approach target to hole {hole.name} and back.")

# --- Main execution: Run only the new functions ---
if __name__ == '__main__':
    create_face_targets()
    create_face_programs()

--- Python program csvimporterLauranewest ---
# This macro can load CSV files from Denso programs in RoboDK.
# Supported types of files are:
#  1-Tool data : Tool.csv
#  2-Work object data: Work.csv
#  3-Target data: P_Var.csv
# This macro can also filter a given targets file

# Type help("robodk.robolink") or help("robodk.robomath") for more information
# Press F5 to run the script
# Visit: http://www.robodk.com/doc/PythonAPI/
# For RoboDK API documentation

import os
import datetime

from robodk.robolink import *  # API to communicate with RoboDK
from robodk.robomath import *  # Robot toolbox
from robodk.robodialogs import *
from robodk.robofileio import *
import robodk.robolinkutils as RDKutils

DEBUG = False

debuglist = []

# Start communication with RoboDK
RDK = Robolink()

# Ask the user to select the robot
ROBOT = RDK.ItemUserPick('Select a robot', ITEM_TYPE_ROBOT)

# Check if the user selected a robot
if not ROBOT.Valid():
    quit()


# Ask the user to select a reference frame and get the active tool
BASE = ROBOT.Parent()
#BASE = RDK.Item('UR10e Base', ITEM_TYPE_FRAME)
#BASE = RDK.ItemUserPick('Select robot base frame', ITEM_TYPE_FRAME)
FRAME = RDK.ItemUserPick('Reference Frame', ITEM_TYPE_FRAME)
FRAMEPOSE = RDKutils.getPoseWrt(FRAME, BASE) #frame pose wrt robot base
TOOL = ROBOT.getLink(ITEM_TYPE_TOOL)
TOOLPOSE = RDKutils.getPoseWrt(TOOL, TOOL.Parent()) #tool pose wrt robot flange

if not FRAME.Valid() or not TOOL.Valid():
    raise Exception("Select appropriate FRAME and TOOL references")


# Function to convert XYZWPR to a pose
# Important! Specify the order of rotation
def xyzwpr_to_pose(xyzwpr):
    x, y, z, rx, ry, rz = xyzwpr
    return point_Zaxis_2_pose([x, y, z], [-rx, -ry, -rz], [0, 0, -1], [0, 1, -1])


csv_file = getOpenFileName(RDK.getParam('PATH_OPENSTATION'))

# Specify file codec
codec = 'utf-8'  #'ISO-8859-1'


# Load P_Var.CSV data as a list of poses, including links to reference and tool frames
def load_targets(strfile):
    csvdata = LoadList(strfile, ',', codec)
    poses = []
    idxs = []
    for i in range(0, len(csvdata)):
        x, y, z, rx, ry, rz = csvdata[i][0:6]
        poses.append(xyzwpr_to_pose([x, y, z, rx, ry, rz]))
        #idxs.append(csvdata[i][6])
        idxs.append(i)

    return poses, idxs


# Load and display Targets from P_Var.CSV in RoboDK
def make_targets(strfile):
    poses, idxs = load_targets(strfile)
    program_name = os.path.basename(strfile)

    for pose, idx in zip(poses, idxs):
        name = 'H-%s-%i' % (program_name, idx)
        target = RDK.Item(name, ITEM_TYPE_TARGET)
        if target.Valid():
            target.Delete()
        target = RDK.AddTarget(name, FRAME, ROBOT)
        target.setPose(pose)
        collision_free(target, idx)

def test_all_configurations(configurations):
    for joints in configurations:

        # turn collision checking off
        RDK.setCollisionActive(COLLISION_OFF)
        if DEBUG:
            is_active = RDK.Command("CollisionActive")
            print(f"collsion active? should be off (0) {is_active}")
            debuglist.append(f"collsion active? should be off (0) {is_active}")

        # move to target
        try:
            ROBOT.MoveJ(joints)
        except TargetReachError:
            continue

        # turn collision checking on, test for collisions
        RDK.setCollisionActive(COLLISION_ON)
        if DEBUG:
            is_active = RDK.Command("CollisionActive")
            print(f"collsion active? should be on (1) {is_active}")
            debuglist.append(f"collsion active? should be on (1) {is_active}")

        collision = RDK.Collisions()
        if DEBUG:
            print(f"collision: {collision}")
            debuglist.append(f"collision: {collision}")

        if collision == 0: #solution found
            break

        collision_items = RDK.CollisionItems()
        if TOOL in collision_items: #no solution possible with current rotation
            break

    try:
        collision
    except NameError:
        collision = -2
        if DEBUG:
            print("Target cannot be reached or is to close to a singularity")
            debuglist.append("Target cannot be reached or is to close to a singularity")

    return collision

def test_issues_point(target, rz):
    if DEBUG:
        print("testing point")
        debuglist.append("testing point")

    # define the rotated position to test for collisions
    target_new_pose = RelTool(target.Pose(), 0,0,0, 0,0,rz)
    possible_robot_configurations = ROBOT.SolveIK_All(target_new_pose, tool=TOOLPOSE, reference=FRAMEPOSE)
    issues_value = test_all_configurations(possible_robot_configurations) # returns 0 if at least one configuration is without issues

    return issues_value, target_new_pose

rotation_direction = "pos"
direction_changes = 0
holes_no_solution = []

def collision_free(target, idx):
    rotation_step = 10
    repmax = 360/rotation_step
    global rotation_direction
    global direction_changes
    s = 0
    rep = 0
    if DEBUG:
        print(f"\nHole {idx}")
        debuglist.append(f"\nHole {idx}")

    issues_value, target_new_pose = test_issues_point(target, 0)
    if DEBUG:
        print(f"issues value: {issues_value}")
        debuglist.append(f"issues value: {issues_value}")

    while issues_value != 0 and s < 100: # s for safety, so it can't go on forever
        if DEBUG:
            print(f"s before: {s}")
            debuglist.append(f"s before: {s}")
            print(f"rep: {rep}")
            debuglist.append(f"rep: {rep}")
            print(f"rotation direction: {rotation_direction}")
            debuglist.append(f"rotation direction: {rotation_direction}")
            print(f"direction changes: {direction_changes}")
            debuglist.append(f"direction changes: {direction_changes}")

        s += 1

        if issues_value == -2 and direction_changes < 2:
			#target unreachable
            if rotation_direction == "pos":
                rotation_direction = "neg"
                direction_changes += 1
                r = -1 #rotation factor to make the rotation negative
            else:
                rotation_direction = "pos"
                direction_changes += 1
                r = 1 #rotation factor to make the rotation positive
            issues_value, target_new_pose = test_issues_point(target, r*rotation_step)
            target.setPose(target_new_pose)

        elif issues_value > 0 and rep < repmax:
			#collision
            RDK.setCollisionActive(COLLISION_OFF)
            if DEBUG:
                is_active = RDK.Command("CollisionActive")
                print(f"collsion active? should be off (0) {is_active}")
                debuglist.append(f"collsion active? should be off (0) {is_active}")

            ROBOT.MoveJ(target.Pose())
            if rotation_direction == "neg":
                r = -1
            elif rotation_direction == "pos":
                r = 1
            issues_value, target_new_pose = test_issues_point(target, r*rotation_step)
            target.setPose(target_new_pose)
            rep += 1

        elif direction_changes >= 2 or rep >= repmax:
            break

        else:
            RDK.ShowMessage(f"Unknown error occured at Hole {idx} while looking for collision free position")
            if DEBUG:
                print(f"Unknown error occured at Hole {idx} while looking for collision free position")
                debuglist.append(f"Unknown error occured at Hole {idx} while looking for collision free position")

    direction_changes = 0
    if issues_value == 0:
        print(f"No issues at Hole {idx}")
        debuglist.append(f"No issues at Hole {idx}")
    elif direction_changes >= 2 or rep >= repmax or s >= 100:
        RDK.ShowMessage(f"No solution found for Hole {idx}", False)
        holes_no_solution.append(idx)
        if DEBUG:
            print(f"No solution found for Hole {idx}")
            debuglist.append(f"No solution found for Hole {idx}")
    else:
        RDK.ShowMessage(f"Unknown error occured at Hole {idx} while looking for collision free position")
        if DEBUG:
            print(f"Unknown error occured at Hole {idx} while looking for collision free position")
            debuglist.append(f"Unknown error occured at Hole {idx} while looking for collision free position")


MAKE_GUI_PROGRAM = True

ROBOT.setFrame(FRAME)
ROBOT.setTool(TOOL)

if RDK.RunMode() == RUNMODE_SIMULATE:
    MAKE_GUI_PROGRAM = True
    # MAKE_GUI_PROGRAM = mbox('Do you want to create a new program? If not, the robot will just move along the targets', 'Yes', 'No')
else:
    # if we run in program generation mode just move the robot
    MAKE_GUI_PROGRAM = False

if MAKE_GUI_PROGRAM:
    RDK.Render(False)  # Faster if we turn render off
    make_targets(csv_file)
else:
    l

RDK.ShowMessage(f"Holes without solution: {holes_no_solution}")

if DEBUG:
    print(f"Holes without solution: {holes_no_solution}")
    debuglist.append(f"Holes without solution: {holes_no_solution}")

    current_time = datetime.datetime.now()
    filename = os.path.splitext(os.path.basename(__file__))
    with open("C:/Users/Laura/Documents/1.Windesheim/Stage/2024/Lectoraat/Deelvragen/2.Targets maken/debugfile.txt", "a") as file:
        file.write("\n\n-----------------------------------------------\n")
        file.write(current_time.strftime("%c"))
        file.write("\n-----------------------------------------------\n")
        for prints in debuglist:
            file.write(prints)
            file.write("\n")
        file.write(holes_no_solution)
        file.write(filename[0])

--- Python program Addmoveshanktoprog ---
from robodk import robolink, robomath

# Connect to RoboDK
RDK = robolink.Robolink()

# Ask the user to select the program to duplicate
orig_prog = RDK.ItemUserPick("Select the program to duplicate", robolink.ITEM_TYPE_PROGRAM)
if not orig_prog.Valid():
    print("No valid program selected.")
    quit()

# Create a new program (a duplicate) with a new name
new_prog_name = "New_" + orig_prog.Name()
new_prog = RDK.AddProgram(new_prog_name)
print("Creating new program:", new_prog.Name())

# Get the number of instructions from the original program
ins_count = orig_prog.InstructionCount()
print("Original program '{}' has {} instructions.".format(orig_prog.Name(), ins_count))

# Iterate over each instruction in the original program
for i in range(ins_count):
    # Retrieve instruction info as a dictionary.
    # Note: Calling setParam(i) with only the index returns the instruction information.
    ins_dict = orig_prog.setParam(i)

    # Try to get the command code string from the instruction dictionary.
    # (Many instructions have a "Code" key that holds the Python command as text.)
    code_line = ins_dict.get("Code", "").strip()
    if not code_line:
        print("Skipping instruction {} because no code is available.".format(i))
        continue

    # Add the instruction to the new program
    print("Adding instruction {}: {}".format(i, code_line))
    new_prog.RunInstruction(code_line, robolink.INSTRUCTION_CALL_PROGRAM)

    # If the instruction contains "FaceTarget" then add two extra moveshank instructions after it.
    if "Face_Target" in code_line:
        print("Detected 'FaceTarget' at instruction {}. Inserting moveshank instructions.".format(i))
        new_prog.RunInstruction('move_shank(20)', robolink.INSTRUCTION_CALL_PROGRAM)
        new_prog.RunInstruction('move_shank(0)', robolink.INSTRUCTION_CALL_PROGRAM)

# Finalize the new program; this applies the modifications
new_prog.Update()
print("New program '{}' created successfully.".format(new_prog.Name()))

--- program Prog20 (robot UR10e) ---
  Set Ref.: CSV Frame
  Set Tool: TCP Schroeftool
  MoveL (Target 36)
  Call Program_Face_-1_0_0
  Call Program_Face_-1_0_0
  MoveL (Target 36)
  MoveL (Target 35)
  MoveJ (Target 37 new)
  MoveL (Target 37 new)
  MoveL (Target 35)
  Call Program_Face_0_-1_1
  MoveL (Target 35)
  Call Program_Face_0_-1_0
  MoveL (Target 35)

--- program Program_Face_-1_0_0 (robot UR10e) ---
  Set Ref.: CSV Frame
  Set Tool: TCP Schroeftool
  MoveL (Target 36)
  MoveL (Face_Target_-1_0_0)
  MoveL (H-12.5_30.0-9)
  MoveL (Face_Target_-1_0_0)
  MoveL (H-12.5_30.0-10)
  MoveL (Face_Target_-1_0_0)
  MoveL (H-12.5_30.0-11)
  MoveL (Face_Target_-1_0_0)
  MoveL (H-12.5_30.0-12)
  MoveL (Face_Target_-1_0_0)
  MoveL (H-12.5_30.0-13)
  MoveL (Face_Target_-1_0_0)
  MoveL (H-12.5_30.0-14)
  MoveL (Face_Target_-1_0_0)
  MoveL (H-12.5_30.0-15)
  MoveL (Face_Target_-1_0_0)
  MoveL (Target 36)

--- program Program_Face_0_0_1 (robot UR10e) ---
  Set Ref.: CSV Frame
  Set Tool: TCP Schroeftool
  MoveL (Face_Target_0_0_1)
  MoveL (H-12.4_20.0-0)
  MoveL (Face_Target_0_0_1)
  MoveL (H-12.4_20.0-1)
  MoveL (Face_Target_0_0_1)
  MoveL (H-12.4_20.0-2)
  MoveL (Face_Target_0_0_1)
  MoveL (H-12.4_20.0-3)
  MoveL (Face_Target_0_0_1)
  MoveL (H-12.4_20.0-4)
  MoveL (Face_Target_0_0_1)
  MoveL (H-12.4_20.0-5)
  MoveL (Face_Target_0_0_1)
  MoveL (H-12.4_20.0-6)
  MoveL (Face_Target_0_0_1)

--- program Program_Face_0_-1_1 (robot UR10e) ---
  Set Ref.: CSV Frame
  Set Tool: TCP Schroeftool
  MoveL (Target 35)
  MoveJ (Target 37 new)
  MoveL (Toolswitch-m8)
  MoveL (Aanlevering-Pos1)
  MoveJ (Target 37 new)
  MoveJ (Target 35)
  MoveL (Face_Target_0_-1_1)
  MoveL (H-12.4_20.0-10)
  Call move_shank(20)
  Call move_shank(0)
  MoveL (Target 35)
  MoveJ (Target 37 new)
  MoveL (Aanlevering-Pos1)
  MoveJ (Target 37 new)
  MoveJ (Target 35)
  MoveL (Face_Target_0_-1_1)
  MoveL (H-12.4_20.0-11)
  Call move_shank(20)
  Call move_shank(0)
  MoveL (Target 35)
  MoveJ (Target 37 new)
  MoveL (Aanlevering-Pos1)
  MoveJ (Target 37 new)
  MoveJ (Target 35)
  MoveL (Face_Target_0_-1_1)
  MoveL (H-12.4_20.0-12)
  Call move_shank(20)
  Call move_shank(0)
  MoveL (Target 35)
  MoveJ (Target 37 new)
  MoveL (Aanlevering-Pos1)
  MoveJ (Target 37 new)
  MoveJ (Target 35)
  MoveL (Face_Target_0_-1_1)
  MoveL (H-12.4_20.0-13)
  Call move_shank(20)
  Call move_shank(0)
  MoveL (Target 35)
  MoveJ (Target 37 new)
  MoveL (Aanlevering-Pos1)
  MoveJ (Target 37 new)
  MoveJ (Target 35)
  MoveL (Face_Target_0_-1_1)
  MoveL (H-12.4_20.0-14)
  Call move_shank(20)
  Call move_shank(0)
  MoveL (Target 35)
  MoveJ (Target 37 new)
  MoveL (Aanlevering-Pos1)
  MoveJ (Target 37 new)
  MoveL (Target 35)
  - Wanneer face target wordt gemaakt, tussen elke gat moet een helicoil opgepakt worden
- manier bedenken om "Aanlevering-Pos1" target te zoeken 
- manier om Toolswitch-m8 target te zoeken
- wanneer de aanlevering of toolswitch benadert wordt moet dat via target 35 -> target 37

wat er nu aangepast moet worden, moet via de approach points benaderd worden 
de flow voor een gat is de volgende Target 35 -> Target 37 -> Oppakken helicoil, dan via hetzelfde route terug gaan, Target 37 -> Target 35 en naar approach. 
voor elke gat moeten er minimaal 5 bewegingen komen

--- program Program_Face_0_-1_0 (robot UR10e) ---
  Set Ref.: CSV Frame
  Set Tool: TCP Schroeftool
  MoveL (Face_Target_0_-1_0)
  MoveL (H-12.4_20.0-18)
  MoveL (Face_Target_0_-1_0)
  MoveL (H-12.4_20.0-19)
  MoveL (Face_Target_0_-1_0)
  MoveL (H-12.4_20.0-20)
  MoveL (Face_Target_0_-1_0)
  MoveL (H-12.4_20.0-21)
  MoveL (Face_Target_0_-1_0)
  MoveL (H-12.4_20.0-22)
  MoveL (Face_Target_0_-1_0)

--- program Prog22 (robot UR10e) ---
  Set Ref.: CSV Frame
  Set Tool: TCP Schroeftool
  MoveL (Target 36)
  MoveL (Target 35)
  MoveJ (Target 37 new)
  MoveL (Toolswitch-m8)
  Call move_shank(20)
  Call move_shank(0)
  MoveL (H-10.2_4-0) -> target Aanlevering-Pos1
  Call move_shank(20)
  Call move_shank(0)
  MoveL (Target 37 new)
